KUKA KRL program: EPS_2_251729_MH1_A_20251114081654.src

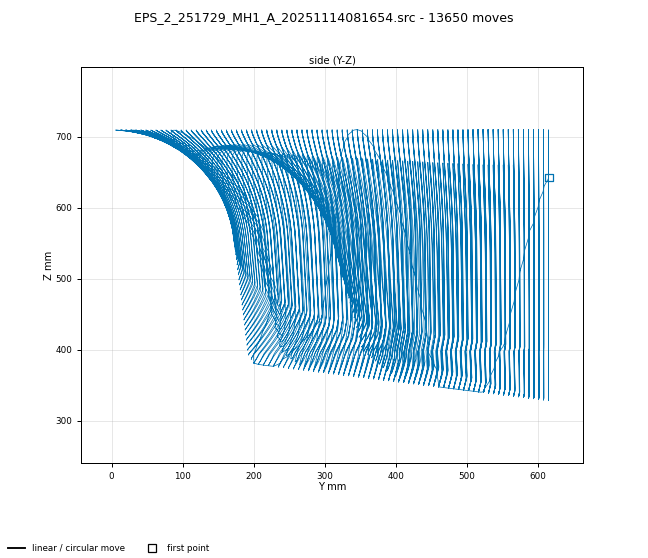
[picture p0: tool path of EPS_2_251729_MH1_A_20251114081654.src, 13650 of 13652 moves have a stored position in this frame; points joined in program order, loops and branches not executed]
&ACCESS RVP
&REL 4
&COMMENT QRS 19112012
&PARAM EDITMASK = *
DEF PART()
EXT BAS (BAS_COMMAND :IN,REAL :IN )
INT I
BAS (#INITMOV,0 )

;KUKA QRS Post kuka4.cps  Date:22-06-2017 !

File_ID=2915

QRS_PRE_INIT()

;Init var - Until changes are made in qrs_pre_init
Outlet_Square_prg=0
Inlet_1_Square_prg=0
Inlet_2_Square_prg=0
Inlet_3_Square_prg=0
Inlet_4_Square_prg=0
Inlet_5_Square_prg=0

Outlet_1={X 0.000, Y 517.920, Z 561.000, B 0.000, E1 0.000 }
Inlet_1={X 0.000, Y 525.500, Z 535.000, B 0.000, E1 90.000 }
Inlet_2={X 0.000, Y 517.920, Z 561.000, B 0.000, E1 180.000 }
Outlet_1_type=299
Inlet_1_type=251
Inlet_2_type=299
;QRS#1=Sidecore dimensions
;QRS#2=300-12" PVC SDR 35
;QRS#3=250-10" PVC SDR 35
;QRS#4=300-12" PVC SDR 35
;QRS#5=
;QRS#6=
;QRS#7=
;QRS#8=
;QRS#9=16M PSX
;QRS#10=14M PSX
;QRS#11=16M PSX
;QRS#12=
;QRS#13=
;QRS#14=
;QRS#15=
;QRS#16=1220x127x991 3,25'
;QRS#17=EPS Height
;QRS#18=710,5
;QRS#19=*
;QRS#20= UPDATED VERSION 22-06-2017
;QRS#21=*
Outlet_Square=0150
Inlet_1_Square=0100
Inlet_2_Square=0150
Inlet_3_Square=0
Inlet_4_Square=0
Inlet_5_Square=0
Mill_Square=1
Outlet_Square_Prg=206
Inlet_1_Square_prg=205
Inlet_2_Square_prg=206

QRS_INIT()

$ADVANCE=5

; T1
PTP {E1 173.418,E2 173.418}
PTP {X 0,Y 615.494,A -85,B 0,C 180,E1 173.418,E2 173.418,E3 0,E4 0,E5 0,E6 0}
QRS_SPEED_INIT()
LIN {X 0,Y 615.494,Z 642.738,A -85,B 0,C 180,E1 173.418,E2 173.418,E3 0,E4 0,E5 0,E6 0} C_VEL
LIN {X 0,Y 615.491,Z 635.744,A -85,B 0,C 180,E1 172.289,E2 172.289} C_VEL
LIN {X 0,Y 615.498,Z 628.27,A -85,B 0,C 180,E1 171.298,E2 171.298} C_VEL
LIN {X 0,Y 615.495,Z 619.291,A -85,B 0,C 180,E1 170.304,E2 170.304} C_VEL
LIN {X 0,Y 615.498,Z 608.204,A -85,B 0,C 180,E1 169.291,E2 169.291} C_VEL
LIN {X 0,Y 615.498,Z 597.279,A -85,B 0,C 180,E1 168.473,E2 168.473} C_VEL
LIN {X 0,Y 615.491,Z 584.981,A -85,B 0,C 180,E1 167.721,E2 167.721} C_VEL
LIN {X 0,Y 615.488,Z 573.143,A -85,B 0,C 180,E1 167.134,E2 167.134} C_VEL
LIN {X 0,Y 615.493,Z 560.215,A -85,B 0,C 180,E1 166.631,E2 166.631} C_VEL
LIN {X 0,Y 615.498,Z 547.234,A -85,B 0,C 180,E1 166.252,E2 166.252} C_VEL
LIN {X 0,Y 615.497,Z 533.996,A -85,B 0,C 180,E1 165.988,E2 165.988} C_VEL
LIN {X 0,Y 615.488,Z 397.614,A -85,B 0,C 180,E1 164.35,E2 164.35} C_VEL
LIN {X 0,Y 615.497,Z 392.889,A -85,B 0,C 180,E1 163.832,E2 163.832} C_VEL
LIN {X 0,Y 615.476,Z 369.093,A -85,B 0,C 180,E1 161.008,E2 161.008} C_VEL
LIN {X 0,Y 615.493,Z 345.922,A -85,B 0,C 180,E1 158.216,E2 158.216} C_VEL
LIN {X 0,Y 615.496,Z 328.786,A -85,B 0,C 180,E1 156.104,E2 156.104} C_VEL
LIN {X 0,Y 615.498,Z 328.434,A -85,B 0,C 180,E1 155.99,E2 155.99} C_VEL
LIN {X 0,Y 615.443,Z 328.325,A -85,B 0,C 180,E1 153.554,E2 153.554} C_VEL
LIN {X 0,Y 615.424,Z 328.324,A -85,B 0,C 180,E1 151.339,E2 151.339} C_VEL
LIN {X 0,Y 615.412,Z 328.324,A -85,B 0,C 180,E1 148.926,E2 148.926} C_VEL
LIN {X 0,Y 615.435,Z 328.323,A -85,B 0,C 180,E1 146.474,E2 146.474} C_VEL
LIN {X 0,Y 615.446,Z 328.325,A -85,B 0,C 180,E1 143.572,E2 143.572} C_VEL
LIN {X 0,Y 615.413,Z 328.324,A -85,B 0,C 180,E1 141.09,E2 141.09} C_VEL
LIN {X 0,Y 615.412,Z 328.324,A -85,B 0,C 180,E1 138.914,E2 138.914} C_VEL
LIN {X 0,Y 615.417,Z 328.324,A -85,B 0,C 180,E1 136.749,E2 136.749} C_VEL
LIN {X 0,Y 615.475,Z 328.323,A -85,B 0,C 180,E1 134.151,E2 134.151} C_VEL
LIN {X 0,Y 615.436,Z 328.324,A -85,B 0,C 180,E1 131.478,E2 131.478} C_VEL
LIN {X 0,Y 615.413,Z 328.324,A -85,B 0,C 180,E1 129.053,E2 129.053} C_VEL
LIN {X 0,Y 615.412,Z 328.324,A -85,B 0,C 180,E1 126.927,E2 126.927} C_VEL
LIN {X 0,Y 615.42,Z 328.324,A -85,B 0,C 180,E1 124.691,E2 124.691} C_VEL
LIN {X 0,Y 615.451,Z 328.323,A -85,B 0,C 180,E1 122.325,E2 122.325} C_VEL
LIN {X 0,Y 615.43,Z 328.324,A -85,B 0,C 180,E1 119.409,E2 119.409} C_VEL
LIN {X 0,Y 615.413,Z 328.324,A -85,B 0,C 180,E1 117.031,E2 117.031} C_VEL
LIN {X 0,Y 615.495,Z 328.571,A -85,B 0,C 180,E1 115.806,E2 115.806} C_VEL
LIN {X 0,Y 615.452,Z 348.722,A -85,B 0,C 180,E1 113.558,E2 113.558} C_VEL
LIN {X 0,Y 615.448,Z 371.548,A -85,B 0,C 180,E1 111.082,E2 111.082} C_VEL
LIN {X 0,Y 615.493,Z 396.288,A -85,B 0,C 180,E1 108.443,E2 108.443} C_VEL
LIN {X 0,Y 615.489,Z 398.972,A -85,B 0,C 180,E1 108.2,E2 108.2} C_VEL
LIN {X 0,Y 615.498,Z 565.217,A -85,B 0,C 180,E1 106.186,E2 106.186} C_VEL
LIN {X 0,Y 615.49,Z 580.613,A -85,B 0,C 180,E1 105.863,E2 105.863} C_VEL
LIN {X 0,Y 615.48,Z 595.975,A -85,B 0,C 180,E1 105.396,E2 105.396} C_VEL
LIN {X 0,Y 615.486,Z 610.66,A -85,B 0,C 180,E1 104.803,E2 104.803} C_VEL
LIN {X 0,Y 615.493,Z 624.629,A -85,B 0,C 180,E1 104.09,E2 104.09} C_VEL
LIN {X 0,Y 615.498,Z 637.489,A -85,B 0,C 180,E1 103.285,E2 103.285} C_VEL
LIN {X 0,Y 615.496,Z 649.742,A -85,B 0,C 180,E1 102.363,E2 102.363} C_VEL
LIN {X 0,Y 615.498,Z 660.897,A -85,B 0,C 180,E1 101.36,E2 101.36} C_VEL
LIN {X 0,Y 615.498,Z 671.702,A -85,B 0,C 180,E1 100.194,E2 100.194} C_VEL
LIN {X 0,Y 615.495,Z 680.684,A -85,B 0,C 180,E1 99.033,E2 99.033} C_VEL
LIN {X 0,Y 615.496,Z 688.117,A -85,B 0,C 180,E1 97.876,E2 97.876} C_VEL
LIN {X 0,Y 615.492,Z 695.052,A -85,B 0,C 180,E1 96.557,E2 96.557} C_VEL
LIN {X 0,Y 615.489,Z 700.498,A -85,B 0,C 180,E1 95.241,E2 95.241} C_VEL
LIN {X 0,Y 615.496,Z 704.619,A -85,B 0,C 180,E1 93.929,E2 93.929} C_VEL
LIN {X 0,Y 615.493,Z 707.525,A -85,B 0,C 180,E1 92.618,E2 92.618} C_VEL
LIN {X 0,Y 615.491,Z 709.276,A -85,B 0,C 180,E1 91.309,E2 91.309} C_VEL
LIN {X 0,Y 615.492,Z 709.884,A -85,B 0,C 180,E1 90,E2 90} C_VEL
LIN {X 0,Y 615.493,Z 709.338,A -85,B 0,C 180,E1 88.692,E2 88.692} C_VEL
LIN {X 0,Y 615.496,Z 707.675,A -85,B 0,C 180,E1 87.382,E2 87.382} C_VEL
LIN {X 0,Y 615.496,Z 704.861,A -85,B 0,C 180,E1 86.072,E2 86.072} C_VEL
LIN {X 0,Y 615.489,Z 700.835,A -85,B 0,C 180,E1 84.759,E2 84.759} C_VEL
LIN {X 0,Y 615.491,Z 695.378,A -85,B 0,C 180,E1 83.42,E2 83.42} C_VEL
LIN {X 0,Y 615.493,Z 688.661,A -85,B 0,C 180,E1 82.125,E2 82.125} C_VEL
LIN {X 0,Y 615.491,Z 680.145,A -85,B 0,C 180,E1 80.801,E2 80.801} C_VEL
LIN {X 0,Y 615.495,Z 671.067,A -85,B 0,C 180,E1 79.64,E2 79.64} C_VEL
LIN {X 0,Y 615.496,Z 661.792,A -85,B 0,C 180,E1 78.64,E2 78.64} C_VEL
LIN {X 0,Y 615.496,Z 649.823,A -85,B 0,C 180,E1 77.554,E2 77.554} C_VEL
LIN {X 0,Y 615.497,Z 637.582,A -85,B 0,C 180,E1 76.631,E2 76.631} C_VEL
LIN {X 0,Y 615.497,Z 624.88,A -85,B 0,C 180,E1 75.835,E2 75.835} C_VEL
LIN {X 0,Y 615.484,Z 610.782,A -85,B 0,C 180,E1 75.113,E2 75.113} C_VEL
LIN {X 0,Y 615.479,Z 596.123,A -85,B 0,C 180,E1 74.519,E2 74.519} C_VEL
LIN {X 0,Y 615.492,Z 581.162,A -85,B 0,C 180,E1 74.062,E2 74.062} C_VEL
LIN {X 0,Y 615.499,Z 565.657,A -85,B 0,C 180,E1 73.732,E2 73.732} C_VEL
LIN {X 0,Y 615.476,Z 447.644,A -85,B 0,C 180,E1 72.301,E2 72.301} C_VEL
LIN {X 0,Y 615.489,Z 398.701,A -85,B 0,C 180,E1 71.699,E2 71.699} C_VEL
LIN {X 0,Y 615.468,Z 374.018,A -85,B 0,C 180,E1 69.094,E2 69.094} C_VEL
LIN {X 0,Y 615.447,Z 351.178,A -85,B 0,C 180,E1 66.62,E2 66.62} C_VEL
LIN {X 0,Y 615.495,Z 328.663,A -85,B 0,C 180,E1 64.126,E2 64.126} C_VEL
LIN {X 0,Y 615.492,Z 328.327,A -85,B 0,C 180,E1 63.921,E2 63.921} C_VEL
LIN {X 0,Y 615.42,Z 328.325,A -85,B 0,C 180,E1 61.339,E2 61.339} C_VEL
LIN {X 0,Y 615.41,Z 328.325,A -85,B 0,C 180,E1 58.926,E2 58.926} C_VEL
LIN {X 0,Y 615.439,Z 328.325,A -85,B 0,C 180,E1 56.473,E2 56.473} C_VEL
LIN {X 0,Y 615.441,Z 328.323,A -85,B 0,C 180,E1 53.572,E2 53.572} C_VEL
LIN {X 0,Y 615.416,Z 328.323,A -85,B 0,C 180,E1 51.09,E2 51.09} C_VEL
LIN {X 0,Y 615.418,Z 328.324,A -85,B 0,C 180,E1 48.913,E2 48.913} C_VEL
LIN {X 0,Y 615.429,Z 328.323,A -85,B 0,C 180,E1 46.75,E2 46.75} C_VEL
LIN {X 0,Y 615.486,Z 328.322,A -85,B 0,C 180,E1 43.997,E2 43.997} C_VEL
LIN {X 0,Y 615.438,Z 328.32,A -85,B 0,C 180,E1 41.478,E2 41.478} C_VEL
LIN {X 0,Y 615.464,Z 328.319,A -85,B 0,C 180,E1 39.752,E2 39.752} C_VEL
LIN {X 0,Y 615.429,Z 328.32,A -85,B 0,C 180,E1 37.246,E2 37.246} C_VEL
LIN {X 0,Y 615.447,Z 328.323,A -85,B 0,C 180,E1 34.695,E2 34.695} C_VEL
LIN {X 0,Y 615.46,Z 328.317,A -85,B 0,C 180,E1 31.687,E2 31.687} C_VEL
LIN {X 0,Y 615.44,Z 328.318,A -85,B 0,C 180,E1 29.409,E2 29.409} C_VEL
LIN {X 0,Y 615.437,Z 328.32,A -85,B 0,C 180,E1 27.036,E2 27.036} C_VEL
LIN {X 0,Y 615.493,Z 328.324,A -85,B 0,C 180,E1 24.272,E2 24.272} C_VEL
LIN {X 0,Y 615.445,Z 328.317,A -85,B 0,C 180,E1 21.434,E2 21.434} C_VEL
LIN {X 0,Y 615.443,Z 328.317,A -85,B 0,C 180,E1 19.339,E2 19.339} C_VEL
LIN {X 0,Y 615.443,Z 328.318,A -85,B 0,C 180,E1 17.272,E2 17.272} C_VEL
LIN {X 0,Y 615.486,Z 328.324,A -85,B 0,C 180,E1 14.549,E2 14.549} C_VEL
LIN {X 0,Y 615.482,Z 328.312,A -85,B 0,C 180,E1 11.861,E2 11.861} C_VEL
LIN {X 0,Y 615.448,Z 328.318,A -85,B 0,C 180,E1 9.199,E2 9.199} C_VEL
LIN {X 0,Y 615.49,Z 328.326,A -85,B 0,C 180,E1 6.557,E2 6.557} C_VEL
LIN {X 0,Y 615.484,Z 328.311,A -85,B 0,C 180,E1 3.929,E2 3.929} C_VEL
LIN {X 0,Y 615.453,Z 328.316,A -85,B 0,C 180,E1 1.309,E2 1.309} C_VEL
LIN {X 0,Y 615.489,Z 328.324,A -85,B 0,C 180,E1 -1.309,E2 -1.309} C_VEL
LIN {X 0,Y 615.49,Z 328.311,A -85,B 0,C 180,E1 -3.928,E2 -3.928} C_VEL
LIN {X 0,Y 615.459,Z 328.314,A -85,B 0,C 180,E1 -6.557,E2 -6.557} C_VEL
LIN {X 0,Y 615.486,Z 328.323,A -85,B 0,C 180,E1 -9.199,E2 -9.199} C_VEL
LIN {X 0,Y 615.493,Z 328.31,A -85,B 0,C 180,E1 -11.861,E2 -11.861} C_VEL
LIN {X 0,Y 615.463,Z 328.314,A -85,B 0,C 180,E1 -14.55,E2 -14.55} C_VEL
LIN {X 0,Y 615.495,Z 328.326,A -85,B 0,C 180,E1 -17.27,E2 -17.27} C_VEL
LIN {X 0,Y 615.487,Z 328.308,A -85,B 0,C 180,E1 -20.033,E2 -20.033} C_VEL
LIN {X 0,Y 615.472,Z 328.319,A -85,B 0,C 180,E1 -22.845,E2 -22.845} C_VEL
LIN {X 0,Y 615.484,Z 328.316,A -85,B 0,C 180,E1 -25.568,E2 -25.568} C_VEL
LIN {X 0,Y 615.486,Z 328.309,A -85,B 0,C 180,E1 -27.915,E2 -27.915} C_VEL
LIN {X 0,Y 615.486,Z 328.308,A -85,B 0,C 180,E1 -30.16,E2 -30.16} C_VEL
LIN {X 0,Y 615.473,Z 328.313,A -85,B 0,C 180,E1 -32.458,E2 -32.458} C_VEL
LIN {X 0,Y 615.475,Z 328.321,A -85,B 0,C 180,E1 -34.816,E2 -34.816} C_VEL
LIN {X 0,Y 615.484,Z 328.322,A -85,B 0,C 180,E1 -37.242,E2 -37.242} C_VEL
LIN {X 0,Y 615.492,Z 328.306,A -85,B 0,C 180,E1 -40.09,E2 -40.09} C_VEL
LIN {X 0,Y 615.489,Z 328.326,A -85,B 0,C 180,E1 -43.047,E2 -43.047} C_VEL
LIN {X 0,Y 615.487,Z 328.307,A -85,B 0,C 180,E1 -46.003,E2 -46.003} C_VEL
LIN {X 0,Y 615.487,Z 328.326,A -85,B 0,C 180,E1 -48.905,E2 -48.905} C_VEL
LIN {X 0,Y 615.486,Z 328.322,A -85,B 0,C 180,E1 -51.096,E2 -51.096} C_VEL
LIN {X 0,Y 615.474,Z 328.313,A -85,B 0,C 180,E1 -53.574,E2 -53.574} C_VEL
LIN {X 0,Y 615.482,Z 328.316,A -85,B 0,C 180,E1 -56.466,E2 -56.466} C_VEL
LIN {X 0,Y 615.479,Z 328.322,A -85,B 0,C 180,E1 -59.08,E2 -59.08} C_VEL
LIN {X 0,Y 615.47,Z 328.313,A -85,B 0,C 180,E1 -61.553,E2 -61.553} C_VEL
LIN {X 0,Y 615.483,Z 328.313,A -85,B 0,C 180,E1 -64.284,E2 -64.284} C_VEL
LIN {X 0,Y 615.498,Z 328.586,A -85,B 0,C 180,E1 -64.937,E2 -64.937} C_VEL
LIN {X 0,Y 615.476,Z 347.018,A -85,B 0,C 180,E1 -66.8,E2 -66.8} C_VEL
LIN {X 0,Y 615.435,Z 372.213,A -85,B 0,C 180,E1 -69.267,E2 -69.267} C_VEL
LIN {X 0,Y 615.496,Z 398.105,A -85,B 0,C 180,E1 -71.742,E2 -71.742} C_VEL
LIN {X 0,Y 615.498,Z 564.923,A -85,B 0,C 180,E1 -73.764,E2 -73.764} C_VEL
LIN {X 0,Y 615.49,Z 580.716,A -85,B 0,C 180,E1 -74.095,E2 -74.095} C_VEL
LIN {X 0,Y 615.477,Z 596.053,A -85,B 0,C 180,E1 -74.562,E2 -74.562} C_VEL
LIN {X 0,Y 615.486,Z 609.755,A -85,B 0,C 180,E1 -75.113,E2 -75.113} C_VEL
LIN {X 0,Y 615.493,Z 624.047,A -85,B 0,C 180,E1 -75.834,E2 -75.834} C_VEL
LIN {X 0,Y 615.497,Z 636.9,A -85,B 0,C 180,E1 -76.631,E2 -76.631} C_VEL
LIN {X 0,Y 615.495,Z 649.256,A -85,B 0,C 180,E1 -77.554,E2 -77.554} C_VEL
LIN {X 0,Y 615.495,Z 659.607,A -85,B 0,C 180,E1 -78.473,E2 -78.473} C_VEL
LIN {X 0,Y 615.494,Z 669.185,A -85,B 0,C 180,E1 -79.473,E2 -79.473} C_VEL
LIN {X 0,Y 615.493,Z 678.578,A -85,B 0,C 180,E1 -80.636,E2 -80.636} C_VEL
LIN {X 0,Y 615.497,Z 686.381,A -85,B 0,C 180,E1 -81.794,E2 -81.794} C_VEL
LIN {X 0,Y 615.494,Z 693.609,A -85,B 0,C 180,E1 -83.102,E2 -83.102} C_VEL
LIN {X 0,Y 615.499,Z 699.437,A -85,B 0,C 180,E1 -84.43,E2 -84.43} C_VEL
LIN {X 0,Y 615.491,Z 702.86,A -85,B 0,C 180,E1 -85.416,E2 -85.416} C_VEL
LIN {X 0,Y 615.493,Z 706.318,A -85,B 0,C 180,E1 -86.727,E2 -86.727} C_VEL
LIN {X 0,Y 615.499,Z 708.593,A -85,B 0,C 180,E1 -88.037,E2 -88.037} C_VEL
LIN {X 0,Y 615.491,Z 709.741,A -85,B 0,C 180,E1 -89.346,E2 -89.346} C_VEL
LIN {X 0,Y 615.491,Z 709.741,A -85,B 0,C 180,E1 -90.654,E2 -90.654} C_VEL
LIN {X 0,Y 615.499,Z 708.593,A -85,B 0,C 180,E1 -91.963,E2 -91.963} C_VEL
LIN {X 0,Y 615.493,Z 706.318,A -85,B 0,C 180,E1 -93.273,E2 -93.273} C_VEL
LIN {X 0,Y 615.491,Z 702.86,A -85,B 0,C 180,E1 -94.585,E2 -94.585} C_VEL
LIN {X 0,Y 615.497,Z 698.142,A -85,B 0,C 180,E1 -95.899,E2 -95.899} C_VEL
LIN {X 0,Y 615.492,Z 692.029,A -85,B 0,C 180,E1 -97.216,E2 -97.216} C_VEL
LIN {X 0,Y 615.49,Z 684.332,A -85,B 0,C 180,E1 -98.537,E2 -98.537} C_VEL
LIN {X 0,Y 615.495,Z 676.113,A -85,B 0,C 180,E1 -99.696,E2 -99.696} C_VEL
LIN {X 0,Y 615.496,Z 665.899,A -85,B 0,C 180,E1 -100.892,E2 -100.892} C_VEL
LIN {X 0,Y 615.496,Z 656.066,A -85,B 0,C 180,E1 -101.861,E2 -101.861} C_VEL
LIN {X 0,Y 615.497,Z 643.946,A -85,B 0,C 180,E1 -102.865,E2 -102.865} C_VEL
LIN {X 0,Y 615.498,Z 631.796,A -85,B 0,C 180,E1 -103.706,E2 -103.706} C_VEL
LIN {X 0,Y 615.48,Z 618.377,A -85,B 0,C 180,E1 -104.473,E2 -104.473} C_VEL
LIN {X 0,Y 615.491,Z 603.845,A -85,B 0,C 180,E1 -105.141,E2 -105.141} C_VEL
LIN {X 0,Y 615.478,Z 589.612,A -85,B 0,C 180,E1 -105.651,E2 -105.651} C_VEL
LIN {X 0,Y 615.5,Z 575.075,A -85,B 0,C 180,E1 -106.037,E2 -106.037} C_VEL
LIN {X 0,Y 615.498,Z 560.297,A -85,B 0,C 180,E1 -106.301,E2 -106.301} C_VEL
LIN {X 0,Y 615.495,Z 398.102,A -85,B 0,C 180,E1 -108.258,E2 -108.258} C_VEL
LIN {X 0,Y 615.435,Z 372.211,A -85,B 0,C 180,E1 -110.733,E2 -110.733} C_VEL
LIN {X 0,Y 615.476,Z 347.016,A -85,B 0,C 180,E1 -113.201,E2 -113.201} C_VEL
LIN {X 0,Y 615.498,Z 328.586,A -85,B 0,C 180,E1 -115.063,E2 -115.063} C_VEL
LIN {X 0,Y 615.482,Z 328.314,A -85,B 0,C 180,E1 -115.716,E2 -115.716} C_VEL
LIN {X 0,Y 615.472,Z 328.314,A -85,B 0,C 180,E1 -118.448,E2 -118.448} C_VEL
LIN {X 0,Y 615.484,Z 328.327,A -85,B 0,C 180,E1 -121.086,E2 -121.086} C_VEL
LIN {X 0,Y 615.493,Z 328.307,A -85,B 0,C 180,E1 -124.022,E2 -124.022} C_VEL
LIN {X 0,Y 615.483,Z 328.326,A -85,B 0,C 180,E1 -126.936,E2 -126.936} C_VEL
LIN {X 0,Y 615.475,Z 328.311,A -85,B 0,C 180,E1 -129.751,E2 -129.751} C_VEL
LIN {X 0,Y 615.489,Z 328.316,A -85,B 0,C 180,E1 -132.353,E2 -132.353} C_VEL
LIN {X 0,Y 615.463,Z 328.32,A -85,B 0,C 180,E1 -135.071,E2 -135.071} C_VEL
LIN {X 0,Y 615.487,Z 328.311,A -85,B 0,C 180,E1 -137.92,E2 -137.92} C_VEL
LIN {X 0,Y 615.491,Z 328.319,A -85,B 0,C 180,E1 -140.25,E2 -140.25} C_VEL
LIN {X 0,Y 615.444,Z 328.32,A -85,B 0,C 180,E1 -143.069,E2 -143.069} C_VEL
LIN {X 0,Y 615.439,Z 328.319,A -85,B 0,C 180,E1 -145.306,E2 -145.306} C_VEL
LIN {X 0,Y 615.457,Z 328.318,A -85,B 0,C 180,E1 -147.674,E2 -147.674} C_VEL
LIN {X 0,Y 615.447,Z 328.324,A -85,B 0,C 180,E1 -150.592,E2 -150.592} C_VEL
LIN {X 0,Y 615.421,Z 328.323,A -85,B 0,C 180,E1 -152.967,E2 -152.967} C_VEL
LIN {X 0,Y 615.416,Z 328.324,A -85,B 0,C 180,E1 -155.005,E2 -155.005} C_VEL
LIN {X 0,Y 615.491,Z 328.47,A -85,B 0,C 180,E1 -156.105,E2 -156.105} C_VEL
LIN {X 0,Y 615.494,Z 328.899,A -85,B 0,C 180,E1 -156.218,E2 -156.218} C_VEL
LIN {X 0,Y 615.48,Z 350.974,A -85,B 0,C 180,E1 -158.919,E2 -158.919} C_VEL
LIN {X 0,Y 615.499,Z 374.313,A -85,B 0,C 180,E1 -161.722,E2 -161.722} C_VEL
LIN {X 0,Y 615.485,Z 397.189,A -85,B 0,C 180,E1 -164.413,E2 -164.413} C_VEL
LIN {X 0,Y 615.486,Z 399.616,A -85,B 0,C 180,E1 -164.477,E2 -164.477} C_VEL
LIN {X 0,Y 615.498,Z 535.161,A -85,B 0,C 180,E1 -166.095,E2 -166.095} C_VEL
LIN {X 0,Y 615.497,Z 548.75,A -85,B 0,C 180,E1 -166.379,E2 -166.379} C_VEL
LIN {X 0,Y 615.495,Z 562.489,A -85,B 0,C 180,E1 -166.799,E2 -166.799} C_VEL
LIN {X 0,Y 615.49,Z 574.901,A -85,B 0,C 180,E1 -167.302,E2 -167.302} C_VEL
LIN {X 0,Y 615.498,Z 587.842,A -85,B 0,C 180,E1 -167.972,E2 -167.972} C_VEL
LIN {X 0,Y 615.499,Z 599.559,A -85,B 0,C 180,E1 -168.724,E2 -168.724} C_VEL
LIN {X 0,Y 615.498,Z 611.226,A -85,B 0,C 180,E1 -169.64,E2 -169.64} C_VEL
LIN {X 0,Y 615.497,Z 621.651,A -85,B 0,C 180,E1 -170.636,E2 -170.636} C_VEL
LIN {X 0,Y 615.496,Z 630.24,A -85,B 0,C 180,E1 -171.629,E2 -171.629} C_VEL
LIN {X 0,Y 615.495,Z 638.453,A -85,B 0,C 180,E1 -172.784,E2 -172.784} C_VEL
LIN {X 0,Y 615.496,Z 644.184,A -85,B 0,C 180,E1 -173.773,E2 -173.773} C_VEL
LIN {X 0,Y 615.494,Z 648.887,A -85,B 0,C 180,E1 -174.759,E2 -174.759} C_VEL
LIN {X 0,Y 615.496,Z 653.757,A -85,B 0,C 180,E1 -176.072,E2 -176.072} C_VEL
LIN {X 0,Y 615.496,Z 657.154,A -85,B 0,C 180,E1 -177.382,E2 -177.382} C_VEL
LIN {X 0,Y 615.493,Z 659.174,A -85,B 0,C 180,E1 -178.691,E2 -178.691} C_VEL
LIN {X 0,Y 615.494,Z 659.884,A -85,B 0,C 180,E1 -180,E2 -180} C_VEL
LIN {X 0,Y 615.49,Z 659.28,A -85,B 0,C 180,E1 -181.309,E2 -181.309} C_VEL
LIN {X 0,Y 615.493,Z 657.35,A -85,B 0,C 180,E1 -182.618,E2 -182.618} C_VEL
LIN {X 0,Y 615.496,Z 654.045,A -85,B 0,C 180,E1 -183.929,E2 -183.929} C_VEL
LIN {X 0,Y 615.496,Z 649.273,A -85,B 0,C 180,E1 -185.241,E2 -185.241} C_VEL
LIN {X 0,Y 615.495,Z 642.874,A -85,B 0,C 180,E1 -186.557,E2 -186.557} C_VEL
LIN {X 0,Y 615.494,Z 642.738,A -85,B 0,C 180,E1 -186.582,E2 -186.582} C_VEL
LIN {X 0,Y 614.823,Z 640.104,A -85,B 0,C 180,E1 -187.065,E2 -187.065} C_VEL
LIN {X 0,Y 611.977,Z 635.518,A -85,B 0,C 180,E1 -187.841,E2 -187.841} C_VEL
LIN {X 0,Y 609.129,Z 630.273,A -85,B 0,C 180,E1 -188.592,E2 -188.592} C_VEL
LIN {X 0,Y 608.47,Z 626.658,A -85,B 0,C 180,E1 -189.033,E2 -189.033} C_VEL
LIN {X 0,Y 608.472,Z 617.861,A -85,B 0,C 180,E1 -189.977,E2 -189.977} C_VEL
LIN {X 0,Y 608.506,Z 606.618,A -85,B 0,C 180,E1 -190.973,E2 -190.973} C_VEL
LIN {X 0,Y 608.535,Z 594.824,A -85,B 0,C 180,E1 -191.829,E2 -191.829} C_VEL
LIN {X 0,Y 608.529,Z 581.908,A -85,B 0,C 180,E1 -192.591,E2 -192.591} C_VEL
LIN {X 0,Y 608.566,Z 568.231,A -85,B 0,C 180,E1 -193.227,E2 -193.227} C_VEL
LIN {X 0,Y 608.607,Z 555.002,A -85,B 0,C 180,E1 -193.694,E2 -193.694} C_VEL
LIN {X 0,Y 608.624,Z 540.476,A -85,B 0,C 180,E1 -194.057,E2 -194.057} C_VEL
LIN {X 0,Y 608.632,Z 525.252,A -85,B 0,C 180,E1 -194.289,E2 -194.289} C_VEL
LIN {X 0,Y 608.58,Z 397.863,A -85,B 0,C 180,E1 -195.822,E2 -195.822} C_VEL
LIN {X 0,Y 608.517,Z 396.622,A -85,B 0,C 180,E1 -195.92,E2 -195.92} C_VEL
LIN {X 0,Y 608.533,Z 373.11,A -85,B 0,C 180,E1 -198.732,E2 -198.732} C_VEL
LIN {X 0,Y 608.598,Z 350.263,A -85,B 0,C 180,E1 -201.509,E2 -201.509} C_VEL
LIN {X 0,Y 608.594,Z 330.064,A -85,B 0,C 180,E1 -204.01,E2 -204.01} C_VEL
LIN {X 0,Y 608.481,Z 329.416,A -85,B 0,C 180,E1 -204.153,E2 -204.153} C_VEL
LIN {X 0,Y 608.389,Z 329.321,A -85,B 0,C 180,E1 -206.777,E2 -206.777} C_VEL
LIN {X 0,Y 608.386,Z 329.32,A -85,B 0,C 180,E1 -209.024,E2 -209.024} C_VEL
LIN {X 0,Y 608.391,Z 329.321,A -85,B 0,C 180,E1 -211.321,E2 -211.321} C_VEL
LIN {X 0,Y 608.426,Z 329.321,A -85,B 0,C 180,E1 -213.728,E2 -213.728} C_VEL
LIN {X 0,Y 608.437,Z 329.325,A -85,B 0,C 180,E1 -216.093,E2 -216.093} C_VEL
LIN {X 0,Y 608.394,Z 329.322,A -85,B 0,C 180,E1 -218.594,E2 -218.594} C_VEL
LIN {X 0,Y 608.434,Z 329.32,A -85,B 0,C 180,E1 -220.327,E2 -220.327} C_VEL
LIN {X 0,Y 608.428,Z 329.321,A -85,B 0,C 180,E1 -222.331,E2 -222.331} C_VEL
LIN {X 0,Y 608.398,Z 329.32,A -85,B 0,C 180,E1 -224.801,E2 -224.801} C_VEL
LIN {X 0,Y 608.384,Z 329.32,A -85,B 0,C 180,E1 -227.034,E2 -227.034} C_VEL
LIN {X 0,Y 608.387,Z 329.321,A -85,B 0,C 180,E1 -228.818,E2 -228.818} C_VEL
LIN {X 0,Y 608.392,Z 329.321,A -85,B 0,C 180,E1 -231.406,E2 -231.406} C_VEL
LIN {X 0,Y 608.442,Z 329.323,A -85,B 0,C 180,E1 -233.955,E2 -233.955} C_VEL
LIN {X 0,Y 608.444,Z 329.319,A -85,B 0,C 180,E1 -236.328,E2 -236.328} C_VEL
LIN {X 0,Y 608.404,Z 329.319,A -85,B 0,C 180,E1 -238.739,E2 -238.739} C_VEL
LIN {X 0,Y 608.387,Z 329.321,A -85,B 0,C 180,E1 -240.976,E2 -240.976} C_VEL
LIN {X 0,Y 608.485,Z 329.424,A -85,B 0,C 180,E1 -243.966,E2 -243.966} C_VEL
LIN {X 0,Y 608.726,Z 333.074,A -85,B 0,C 180,E1 -244.418,E2 -244.418} C_VEL
LIN {X 0,Y 608.615,Z 356.881,A -85,B 0,C 180,E1 -247.062,E2 -247.062} C_VEL
LIN {X 0,Y 608.608,Z 382.966,A -85,B 0,C 180,E1 -249.907,E2 -249.907} C_VEL
LIN {X 0,Y 608.603,Z 398.536,A -85,B 0,C 180,E1 -251.566,E2 -251.566} C_VEL
LIN {X 0,Y 608.765,Z 403.562,A -85,B 0,C 180,E1 -251.653,E2 -251.653} C_VEL
LIN {X 0,Y 608.699,Z 565.25,A -85,B 0,C 180,E1 -253.629,E2 -253.629} C_VEL
LIN {X 0,Y 608.651,Z 580.634,A -85,B 0,C 180,E1 -253.954,E2 -253.954} C_VEL
LIN {X 0,Y 608.61,Z 595.973,A -85,B 0,C 180,E1 -254.426,E2 -254.426} C_VEL
LIN {X 0,Y 608.584,Z 610.657,A -85,B 0,C 180,E1 -255.025,E2 -255.025} C_VEL
LIN {X 0,Y 608.571,Z 624.436,A -85,B 0,C 180,E1 -255.735,E2 -255.735} C_VEL
LIN {X 0,Y 608.548,Z 637.545,A -85,B 0,C 180,E1 -256.56,E2 -256.56} C_VEL
LIN {X 0,Y 608.505,Z 649.836,A -85,B 0,C 180,E1 -257.493,E2 -257.493} C_VEL
LIN {X 0,Y 608.497,Z 661.046,A -85,B 0,C 180,E1 -258.508,E2 -258.508} C_VEL
LIN {X 0,Y 608.477,Z 671.931,A -85,B 0,C 180,E1 -259.687,E2 -259.687} C_VEL
LIN {X 0,Y 608.469,Z 680.979,A -85,B 0,C 180,E1 -260.862,E2 -260.862} C_VEL
LIN {X 0,Y 608.46,Z 688.478,A -85,B 0,C 180,E1 -262.033,E2 -262.033} C_VEL
LIN {X 0,Y 608.445,Z 695.629,A -85,B 0,C 180,E1 -263.397,E2 -263.397} C_VEL
LIN {X 0,Y 608.435,Z 700.994,A -85,B 0,C 180,E1 -264.698,E2 -264.698} C_VEL
LIN {X 0,Y 608.432,Z 705.166,A -85,B 0,C 180,E1 -266.026,E2 -266.026} C_VEL
LIN {X 0,Y 608.421,Z 708.11,A -85,B 0,C 180,E1 -267.352,E2 -267.352} C_VEL
LIN {X 0,Y 608.444,Z 709.881,A -85,B 0,C 180,E1 -268.676,E2 -268.676} C_VEL
LIN {X 0,Y 608.432,Z 710.495,A -85,B 0,C 180,E1 -270,E2 -270} C_VEL
LIN {X 0,Y 608.445,Z 709.945,A -85,B 0,C 180,E1 -271.324,E2 -271.324} C_VEL
LIN {X 0,Y 608.424,Z 708.26,A -85,B 0,C 180,E1 -272.648,E2 -272.648} C_VEL
LIN {X 0,Y 608.432,Z 705.407,A -85,B 0,C 180,E1 -273.974,E2 -273.974} C_VEL
LIN {X 0,Y 608.435,Z 701.33,A -85,B 0,C 180,E1 -275.302,E2 -275.302} C_VEL
LIN {X 0,Y 608.446,Z 695.922,A -85,B 0,C 180,E1 -276.633,E2 -276.633} C_VEL
LIN {X 0,Y 608.458,Z 689.021,A -85,B 0,C 180,E1 -277.967,E2 -277.967} C_VEL
LIN {X 0,Y 608.466,Z 681.592,A -85,B 0,C 180,E1 -279.138,E2 -279.138} C_VEL
LIN {X 0,Y 608.477,Z 672.661,A -85,B 0,C 180,E1 -280.313,E2 -280.313} C_VEL
LIN {X 0,Y 608.496,Z 661.949,A -85,B 0,C 180,E1 -281.492,E2 -281.492} C_VEL
LIN {X 0,Y 608.513,Z 649.902,A -85,B 0,C 180,E1 -282.591,E2 -282.591} C_VEL
LIN {X 0,Y 608.543,Z 637.621,A -85,B 0,C 180,E1 -283.525,E2 -283.525} C_VEL
LIN {X 0,Y 608.585,Z 624.675,A -85,B 0,C 180,E1 -284.342,E2 -284.342} C_VEL
LIN {X 0,Y 608.585,Z 610.758,A -85,B 0,C 180,E1 -285.06,E2 -285.06} C_VEL
LIN {X 0,Y 608.631,Z 596.089,A -85,B 0,C 180,E1 -285.659,E2 -285.659} C_VEL
LIN {X 0,Y 608.67,Z 580.52,A -85,B 0,C 180,E1 -286.138,E2 -286.138} C_VEL
LIN {X 0,Y 608.696,Z 565.068,A -85,B 0,C 180,E1 -286.464,E2 -286.464} C_VEL
LIN {X 0,Y 608.683,Z 399.384,A -85,B 0,C 180,E1 -288.492,E2 -288.492} C_VEL
LIN {X 0,Y 608.566,Z 398.143,A -85,B 0,C 180,E1 -288.556,E2 -288.556} C_VEL
LIN {X 0,Y 608.575,Z 374.013,A -85,B 0,C 180,E1 -291.154,E2 -291.154} C_VEL
LIN {X 0,Y 608.614,Z 352.804,A -85,B 0,C 180,E1 -293.478,E2 -293.478} C_VEL
LIN {X 0,Y 608.727,Z 331.079,A -85,B 0,C 180,E1 -295.897,E2 -295.897} C_VEL
LIN {X 0,Y 608.474,Z 329.367,A -85,B 0,C 180,E1 -296.149,E2 -296.149} C_VEL
LIN {X 0,Y 608.383,Z 329.321,A -85,B 0,C 180,E1 -299.024,E2 -299.024} C_VEL
LIN {X 0,Y 608.405,Z 329.32,A -85,B 0,C 180,E1 -301.32,E2 -301.32} C_VEL
LIN {X 0,Y 608.424,Z 329.323,A -85,B 0,C 180,E1 -303.728,E2 -303.728} C_VEL
LIN {X 0,Y 608.438,Z 329.322,A -85,B 0,C 180,E1 -306.093,E2 -306.093} C_VEL
LIN {X 0,Y 608.395,Z 329.321,A -85,B 0,C 180,E1 -308.594,E2 -308.594} C_VEL
LIN {X 0,Y 608.392,Z 329.321,A -85,B 0,C 180,E1 -311.182,E2 -311.182} C_VEL
LIN {X 0,Y 608.461,Z 329.322,A -85,B 0,C 180,E1 -313.87,E2 -313.87} C_VEL
LIN {X 0,Y 608.422,Z 329.316,A -85,B 0,C 180,E1 -316.696,E2 -316.696} C_VEL
LIN {X 0,Y 608.396,Z 329.319,A -85,B 0,C 180,E1 -318.818,E2 -318.818} C_VEL
LIN {X 0,Y 608.407,Z 329.322,A -85,B 0,C 180,E1 -321.407,E2 -321.407} C_VEL
LIN {X 0,Y 608.444,Z 329.321,A -85,B 0,C 180,E1 -323.955,E2 -323.955} C_VEL
LIN {X 0,Y 608.443,Z 329.315,A -85,B 0,C 180,E1 -326.328,E2 -326.328} C_VEL
LIN {X 0,Y 608.428,Z 329.315,A -85,B 0,C 180,E1 -328.735,E2 -328.735} C_VEL
LIN {X 0,Y 608.457,Z 329.317,A -85,B 0,C 180,E1 -331.383,E2 -331.383} C_VEL
LIN {X 0,Y 608.449,Z 329.314,A -85,B 0,C 180,E1 -334.284,E2 -334.284} C_VEL
LIN {X 0,Y 608.46,Z 329.314,A -85,B 0,C 180,E1 -336.155,E2 -336.155} C_VEL
LIN {X 0,Y 608.449,Z 329.314,A -85,B 0,C 180,E1 -338.308,E2 -338.308} C_VEL
LIN {X 0,Y 608.441,Z 329.317,A -85,B 0,C 180,E1 -341.13,E2 -341.13} C_VEL
LIN {X 0,Y 608.461,Z 329.316,A -85,B 0,C 180,E1 -343.906,E2 -343.906} C_VEL
LIN {X 0,Y 608.434,Z 329.315,A -85,B 0,C 180,E1 -346.643,E2 -346.643} C_VEL
LIN {X 0,Y 608.456,Z 329.319,A -85,B 0,C 180,E1 -349.35,E2 -349.35} C_VEL
LIN {X 0,Y 608.475,Z 329.312,A -85,B 0,C 180,E1 -352.033,E2 -352.033} C_VEL
LIN {X 0,Y 608.435,Z 329.315,A -85,B 0,C 180,E1 -354.698,E2 -354.698} C_VEL
LIN {X 0,Y 608.481,Z 329.318,A -85,B 0,C 180,E1 -357.352,E2 -357.352} C_VEL
LIN {X 0,Y 608.477,Z 329.311,A -85,B 0,C 180,E1 -360,E2 -360} C_VEL
LIN {X 0,Y 608.451,Z 329.313,A -85,B 0,C 180,E1 -362.648,E2 -362.648} C_VEL
LIN {X 0,Y 608.466,Z 329.32,A -85,B 0,C 180,E1 -365.302,E2 -365.302} C_VEL
LIN {X 0,Y 608.479,Z 329.31,A -85,B 0,C 180,E1 -367.967,E2 -367.967} C_VEL
LIN {X 0,Y 608.443,Z 329.315,A -85,B 0,C 180,E1 -370.65,E2 -370.65} C_VEL
LIN {X 0,Y 608.468,Z 329.32,A -85,B 0,C 180,E1 -373.356,E2 -373.356} C_VEL
LIN {X 0,Y 608.456,Z 329.312,A -85,B 0,C 180,E1 -376.094,E2 -376.094} C_VEL
LIN {X 0,Y 608.449,Z 329.317,A -85,B 0,C 180,E1 -378.87,E2 -378.87} C_VEL
LIN {X 0,Y 608.47,Z 329.313,A -85,B 0,C 180,E1 -381.691,E2 -381.691} C_VEL
LIN {X 0,Y 608.448,Z 329.314,A -85,B 0,C 180,E1 -384.571,E2 -384.571} C_VEL
LIN {X 0,Y 608.481,Z 329.319,A -85,B 0,C 180,E1 -387.208,E2 -387.208} C_VEL
LIN {X 0,Y 608.468,Z 329.31,A -85,B 0,C 180,E1 -389.972,E2 -389.972} C_VEL
LIN {X 0,Y 608.452,Z 329.319,A -85,B 0,C 180,E1 -392.88,E2 -392.88} C_VEL
LIN {X 0,Y 608.437,Z 329.322,A -85,B 0,C 180,E1 -395.278,E2 -395.278} C_VEL
LIN {X 0,Y 608.468,Z 329.311,A -85,B 0,C 180,E1 -397.746,E2 -397.746} C_VEL
LIN {X 0,Y 608.451,Z 329.313,A -85,B 0,C 180,E1 -400.329,E2 -400.329} C_VEL
LIN {X 0,Y 608.454,Z 329.322,A -85,B 0,C 180,E1 -402.96,E2 -402.96} C_VEL
LIN {X 0,Y 608.458,Z 329.312,A -85,B 0,C 180,E1 -405.736,E2 -405.736} C_VEL
LIN {X 0,Y 608.459,Z 329.317,A -85,B 0,C 180,E1 -408.658,E2 -408.658} C_VEL
LIN {X 0,Y 608.469,Z 329.313,A -85,B 0,C 180,E1 -411.412,E2 -411.412} C_VEL
LIN {X 0,Y 608.447,Z 329.313,A -85,B 0,C 180,E1 -413.954,E2 -413.954} C_VEL
LIN {X 0,Y 608.463,Z 329.313,A -85,B 0,C 180,E1 -416.329,E2 -416.329} C_VEL
LIN {X 0,Y 608.478,Z 329.318,A -85,B 0,C 180,E1 -418.728,E2 -418.728} C_VEL
LIN {X 0,Y 608.459,Z 329.314,A -85,B 0,C 180,E1 -421.382,E2 -421.382} C_VEL
LIN {X 0,Y 608.437,Z 329.316,A -85,B 0,C 180,E1 -423.964,E2 -423.964} C_VEL
LIN {X 0,Y 608.498,Z 329.481,A -85,B 0,C 180,E1 -424.724,E2 -424.724} C_VEL
LIN {X 0,Y 608.739,Z 332.621,A -85,B 0,C 180,E1 -425.077,E2 -425.077} C_VEL
LIN {X 0,Y 608.662,Z 359.615,A -85,B 0,C 180,E1 -427.781,E2 -427.781} C_VEL
LIN {X 0,Y 608.563,Z 388.409,A -85,B 0,C 180,E1 -430.609,E2 -430.609} C_VEL
LIN {X 0,Y 608.627,Z 398.103,A -85,B 0,C 180,E1 -431.529,E2 -431.529} C_VEL
LIN {X 0,Y 608.702,Z 510.075,A -85,B 0,C 180,E1 -432.899,E2 -432.899} C_VEL
LIN {X 0,Y 608.676,Z 565.864,A -85,B 0,C 180,E1 -433.594,E2 -433.594} C_VEL
LIN {X 0,Y 608.656,Z 581.491,A -85,B 0,C 180,E1 -433.933,E2 -433.933} C_VEL
LIN {X 0,Y 608.617,Z 596.051,A -85,B 0,C 180,E1 -434.383,E2 -434.383} C_VEL
LIN {X 0,Y 608.602,Z 609.758,A -85,B 0,C 180,E1 -434.94,E2 -434.94} C_VEL
LIN {X 0,Y 608.573,Z 623.238,A -85,B 0,C 180,E1 -435.624,E2 -435.624} C_VEL
LIN {X 0,Y 608.554,Z 635.665,A -85,B 0,C 180,E1 -436.39,E2 -436.39} C_VEL
LIN {X 0,Y 608.528,Z 648.284,A -85,B 0,C 180,E1 -437.324,E2 -437.324} C_VEL
LIN {X 0,Y 608.496,Z 659.748,A -85,B 0,C 180,E1 -438.339,E2 -438.339} C_VEL
LIN {X 0,Y 608.475,Z 669.389,A -85,B 0,C 180,E1 -439.35,E2 -439.35} C_VEL
LIN {X 0,Y 608.476,Z 678.854,A -85,B 0,C 180,E1 -440.527,E2 -440.527} C_VEL
LIN {X 0,Y 608.456,Z 686.73,A -85,B 0,C 180,E1 -441.699,E2 -441.699} C_VEL
LIN {X 0,Y 608.439,Z 694.088,A -85,B 0,C 180,E1 -443.034,E2 -443.034} C_VEL
LIN {X 0,Y 608.45,Z 699.924,A -85,B 0,C 180,E1 -444.366,E2 -444.366} C_VEL
LIN {X 0,Y 608.427,Z 703.383,A -85,B 0,C 180,E1 -445.362,E2 -445.362} C_VEL
LIN {X 0,Y 608.421,Z 706.886,A -85,B 0,C 180,E1 -446.689,E2 -446.689} C_VEL
LIN {X 0,Y 608.444,Z 709.191,A -85,B 0,C 180,E1 -448.014,E2 -448.014} C_VEL
LIN {X 0,Y 608.434,Z 710.351,A -85,B 0,C 180,E1 -449.338,E2 -449.338} C_VEL
LIN {X 0,Y 608.434,Z 710.351,A -85,B 0,C 180,E1 -450.662,E2 -450.662} C_VEL
LIN {X 0,Y 608.444,Z 709.191,A -85,B 0,C 180,E1 -451.986,E2 -451.986} C_VEL
LIN {X 0,Y 608.421,Z 706.885,A -85,B 0,C 180,E1 -453.311,E2 -453.311} C_VEL
LIN {X 0,Y 608.427,Z 703.382,A -85,B 0,C 180,E1 -454.638,E2 -454.638} C_VEL
LIN {X 0,Y 608.435,Z 698.607,A -85,B 0,C 180,E1 -455.967,E2 -455.967} C_VEL
LIN {X 0,Y 608.456,Z 692.425,A -85,B 0,C 180,E1 -457.3,E2 -457.3} C_VEL
LIN {X 0,Y 608.465,Z 684.653,A -85,B 0,C 180,E1 -458.636,E2 -458.636} C_VEL
LIN {X 0,Y 608.471,Z 676.369,A -85,B 0,C 180,E1 -459.809,E2 -459.809} C_VEL
LIN {X 0,Y 608.492,Z 665.651,A -85,B 0,C 180,E1 -461.063,E2 -461.063} C_VEL
LIN {X 0,Y 608.523,Z 654.273,A -85,B 0,C 180,E1 -462.168,E2 -462.168} C_VEL
LIN {X 0,Y 608.547,Z 642.852,A -85,B 0,C 180,E1 -463.1,E2 -463.1} C_VEL
LIN {X 0,Y 608.563,Z 630.445,A -85,B 0,C 180,E1 -463.95,E2 -463.95} C_VEL
LIN {X 0,Y 608.564,Z 616.856,A -85,B 0,C 180,E1 -464.718,E2 -464.718} C_VEL
LIN {X 0,Y 608.629,Z 602.788,A -85,B 0,C 180,E1 -465.359,E2 -465.359} C_VEL
LIN {X 0,Y 608.634,Z 588.297,A -85,B 0,C 180,E1 -465.874,E2 -465.874} C_VEL
LIN {X 0,Y 608.676,Z 572.925,A -85,B 0,C 180,E1 -466.272,E2 -466.272} C_VEL
LIN {X 0,Y 608.702,Z 557.273,A -85,B 0,C 180,E1 -466.531,E2 -466.531} C_VEL
LIN {X 0,Y 608.637,Z 398.248,A -85,B 0,C 180,E1 -468.466,E2 -468.466} C_VEL
LIN {X 0,Y 608.564,Z 388.407,A -85,B 0,C 180,E1 -469.392,E2 -469.392} C_VEL
LIN {X 0,Y 608.662,Z 359.614,A -85,B 0,C 180,E1 -472.219,E2 -472.219} C_VEL
LIN {X 0,Y 608.74,Z 332.619,A -85,B 0,C 180,E1 -474.923,E2 -474.923} C_VEL
LIN {X 0,Y 608.501,Z 329.48,A -85,B 0,C 180,E1 -475.276,E2 -475.276} C_VEL
LIN {X 0,Y 608.451,Z 329.317,A -85,B 0,C 180,E1 -477.518,E2 -477.518} C_VEL
LIN {X 0,Y 608.468,Z 329.311,A -85,B 0,C 180,E1 -479.972,E2 -479.972} C_VEL
LIN {X 0,Y 608.452,Z 329.322,A -85,B 0,C 180,E1 -482.88,E2 -482.88} C_VEL
LIN {X 0,Y 608.439,Z 329.319,A -85,B 0,C 180,E1 -485.278,E2 -485.278} C_VEL
LIN {X 0,Y 608.466,Z 329.311,A -85,B 0,C 180,E1 -487.747,E2 -487.747} C_VEL
LIN {X 0,Y 608.456,Z 329.316,A -85,B 0,C 180,E1 -490.329,E2 -490.329} C_VEL
LIN {X 0,Y 608.439,Z 329.32,A -85,B 0,C 180,E1 -492.961,E2 -492.961} C_VEL
LIN {X 0,Y 608.451,Z 329.313,A -85,B 0,C 180,E1 -495.737,E2 -495.737} C_VEL
LIN {X 0,Y 608.458,Z 329.32,A -85,B 0,C 180,E1 -498.658,E2 -498.658} C_VEL
LIN {X 0,Y 608.459,Z 329.313,A -85,B 0,C 180,E1 -501.761,E2 -501.761} C_VEL
LIN {X 0,Y 608.432,Z 329.32,A -85,B 0,C 180,E1 -504.722,E2 -504.722} C_VEL
LIN {X 0,Y 608.425,Z 329.317,A -85,B 0,C 180,E1 -507.119,E2 -507.119} C_VEL
LIN {X 0,Y 608.471,Z 329.318,A -85,B 0,C 180,E1 -510.028,E2 -510.028} C_VEL
LIN {X 0,Y 608.409,Z 329.32,A -85,B 0,C 180,E1 -512.806,E2 -512.806} C_VEL
LIN {X 0,Y 608.415,Z 329.32,A -85,B 0,C 180,E1 -515.427,E2 -515.427} C_VEL
LIN {X 0,Y 608.497,Z 329.479,A -85,B 0,C 180,E1 -515.968,E2 -515.968} C_VEL
LIN {X 0,Y 608.63,Z 332.158,A -85,B 0,C 180,E1 -516.343,E2 -516.343} C_VEL
LIN {X 0,Y 608.576,Z 353.874,A -85,B 0,C 180,E1 -519.023,E2 -519.023} C_VEL
LIN {X 0,Y 608.563,Z 377.039,A -85,B 0,C 180,E1 -521.832,E2 -521.832} C_VEL
LIN {X 0,Y 608.532,Z 397.518,A -85,B 0,C 180,E1 -524.252,E2 -524.252} C_VEL
LIN {X 0,Y 608.661,Z 408.603,A -85,B 0,C 180,E1 -524.406,E2 -524.406} C_VEL
LIN {X 0,Y 608.608,Z 535.991,A -85,B 0,C 180,E1 -525.949,E2 -525.949} C_VEL
LIN {X 0,Y 608.613,Z 550.31,A -85,B 0,C 180,E1 -526.264,E2 -526.264} C_VEL
LIN {X 0,Y 608.585,Z 563.648,A -85,B 0,C 180,E1 -526.689,E2 -526.689} C_VEL
LIN {X 0,Y 608.538,Z 576.702,A -85,B 0,C 180,E1 -527.24,E2 -527.24} C_VEL
LIN {X 0,Y 608.538,Z 589.345,A -85,B 0,C 180,E1 -527.917,E2 -527.917} C_VEL
LIN {X 0,Y 608.499,Z 600.848,A -85,B 0,C 180,E1 -528.677,E2 -528.677} C_VEL
LIN {X 0,Y 608.495,Z 611.415,A -85,B 0,C 180,E1 -529.519,E2 -529.519} C_VEL
LIN {X 0,Y 608.48,Z 621.899,A -85,B 0,C 180,E1 -530.527,E2 -530.527} C_VEL
LIN {X 0,Y 608.463,Z 630.551,A -85,B 0,C 180,E1 -531.531,E2 -531.531} C_VEL
LIN {X 0,Y 608.46,Z 638.838,A -85,B 0,C 180,E1 -532.701,E2 -532.701} C_VEL
LIN {X 0,Y 608.443,Z 645.325,A -85,B 0,C 180,E1 -533.831,E2 -533.831} C_VEL
LIN {X 0,Y 608.435,Z 650.787,A -85,B 0,C 180,E1 -535.03,E2 -535.03} C_VEL
LIN {X 0,Y 608.434,Z 654.297,A -85,B 0,C 180,E1 -536.026,E2 -536.026} C_VEL
LIN {X 0,Y 608.424,Z 657.734,A -85,B 0,C 180,E1 -537.352,E2 -537.352} C_VEL
LIN {X 0,Y 608.446,Z 659.778,A -85,B 0,C 180,E1 -538.676,E2 -538.676} C_VEL
LIN {X 0,Y 608.434,Z 660.495,A -85,B 0,C 180,E1 -540,E2 -540} C_VEL
LIN {X 0,Y 608.443,Z 659.881,A -85,B 0,C 180,E1 -541.324,E2 -541.324} C_VEL
LIN {X 0,Y 608.421,Z 657.928,A -85,B 0,C 180,E1 -542.648,E2 -542.648} C_VEL
LIN {X 0,Y 608.434,Z 654.585,A -85,B 0,C 180,E1 -543.974,E2 -543.974} C_VEL
LIN {X 0,Y 608.44,Z 649.76,A -85,B 0,C 180,E1 -545.302,E2 -545.302} C_VEL
LIN {X 0,Y 608.442,Z 643.433,A -85,B 0,C 180,E1 -546.608,E2 -546.608} C_VEL
LIN {X 0,Y 608.451,Z 636.1,A -85,B 0,C 180,E1 -547.8,E2 -547.8} C_VEL
LIN {X 0,Y 608.476,Z 628.56,A -85,B 0,C 180,E1 -548.803,E2 -548.803} C_VEL
LIN {X 0,Y 608.47,Z 626.658,A -85,B 0,C 180,E1 -549.033,E2 -549.033} C_VEL
LIN {X 0,Y 607.811,Z 622.971,A -85,B 0,C 180,E1 -549.46,E2 -549.46} C_VEL
LIN {X 0,Y 604.982,Z 616.737,A -85,B 0,C 180,E1 -550.142,E2 -550.142} C_VEL
LIN {X 0,Y 602.152,Z 610.165,A -85,B 0,C 180,E1 -550.794,E2 -550.794} C_VEL
LIN {X 0,Y 601.494,Z 605.791,A -85,B 0,C 180,E1 -551.169,E2 -551.169} C_VEL
LIN {X 0,Y 601.531,Z 594.814,A -85,B 0,C 180,E1 -551.969,E2 -551.969} C_VEL
LIN {X 0,Y 601.571,Z 581.905,A -85,B 0,C 180,E1 -552.739,E2 -552.739} C_VEL
LIN {X 0,Y 601.64,Z 568.218,A -85,B 0,C 180,E1 -553.382,E2 -553.382} C_VEL
LIN {X 0,Y 601.691,Z 553.909,A -85,B 0,C 180,E1 -553.886,E2 -553.886} C_VEL
LIN {X 0,Y 601.721,Z 539.295,A -85,B 0,C 180,E1 -554.244,E2 -554.244} C_VEL
LIN {X 0,Y 601.77,Z 520.884,A -85,B 0,C 180,E1 -554.508,E2 -554.508} C_VEL
LIN {X 0,Y 601.679,Z 398.345,A -85,B 0,C 180,E1 -555.997,E2 -555.997} C_VEL
LIN {X 0,Y 601.546,Z 397.014,A -85,B 0,C 180,E1 -556.066,E2 -556.066} C_VEL
LIN {X 0,Y 601.609,Z 373.797,A -85,B 0,C 180,E1 -558.872,E2 -558.872} C_VEL
LIN {X 0,Y 601.704,Z 351.707,A -85,B 0,C 180,E1 -561.588,E2 -561.588} C_VEL
LIN {X 0,Y 601.772,Z 332.874,A -85,B 0,C 180,E1 -563.944,E2 -563.944} C_VEL
LIN {X 0,Y 601.432,Z 330.339,A -85,B 0,C 180,E1 -564.317,E2 -564.317} C_VEL
LIN {X 0,Y 601.362,Z 330.196,A -85,B 0,C 180,E1 -567.116,E2 -567.116} C_VEL
LIN {X 0,Y 601.403,Z 330.2,A -85,B 0,C 180,E1 -570.165,E2 -570.165} C_VEL
LIN {X 0,Y 601.384,Z 330.194,A -85,B 0,C 180,E1 -572.71,E2 -572.71} C_VEL
LIN {X 0,Y 601.345,Z 330.198,A -85,B 0,C 180,E1 -575.105,E2 -575.105} C_VEL
LIN {X 0,Y 601.38,Z 330.195,A -85,B 0,C 180,E1 -577.423,E2 -577.423} C_VEL
LIN {X 0,Y 601.393,Z 330.202,A -85,B 0,C 180,E1 -579.997,E2 -579.997} C_VEL
LIN {X 0,Y 601.35,Z 330.198,A -85,B 0,C 180,E1 -582.676,E2 -582.676} C_VEL
LIN {X 0,Y 601.371,Z 330.198,A -85,B 0,C 180,E1 -584.53,E2 -584.53} C_VEL
LIN {X 0,Y 601.401,Z 330.194,A -85,B 0,C 180,E1 -586.43,E2 -586.43} C_VEL
LIN {X 0,Y 601.349,Z 330.197,A -85,B 0,C 180,E1 -589.12,E2 -589.12} C_VEL
LIN {X 0,Y 601.373,Z 330.199,A -85,B 0,C 180,E1 -591.728,E2 -591.728} C_VEL
LIN {X 0,Y 601.372,Z 330.202,A -85,B 0,C 180,E1 -594.244,E2 -594.244} C_VEL
LIN {X 0,Y 601.378,Z 330.195,A -85,B 0,C 180,E1 -596.683,E2 -596.683} C_VEL
LIN {X 0,Y 601.369,Z 330.195,A -85,B 0,C 180,E1 -599.055,E2 -599.055} C_VEL
LIN {X 0,Y 601.358,Z 330.198,A -85,B 0,C 180,E1 -601.369,E2 -601.369} C_VEL
LIN {X 0,Y 601.449,Z 330.416,A -85,B 0,C 180,E1 -603.768,E2 -603.768} C_VEL
LIN {X 0,Y 601.959,Z 333.691,A -85,B 0,C 180,E1 -604.179,E2 -604.179} C_VEL
LIN {X 0,Y 601.811,Z 355.254,A -85,B 0,C 180,E1 -606.606,E2 -606.606} C_VEL
LIN {X 0,Y 601.729,Z 380.287,A -85,B 0,C 180,E1 -609.373,E2 -609.373} C_VEL
LIN {X 0,Y 601.687,Z 398.665,A -85,B 0,C 180,E1 -611.354,E2 -611.354} C_VEL
LIN {X 0,Y 602.025,Z 402.637,A -85,B 0,C 180,E1 -611.429,E2 -611.429} C_VEL
LIN {X 0,Y 601.895,Z 564.61,A -85,B 0,C 180,E1 -613.429,E2 -613.429} C_VEL
LIN {X 0,Y 601.847,Z 579.769,A -85,B 0,C 180,E1 -613.746,E2 -613.746} C_VEL
LIN {X 0,Y 601.774,Z 594.765,A -85,B 0,C 180,E1 -614.201,E2 -614.201} C_VEL
LIN {X 0,Y 601.712,Z 608.732,A -85,B 0,C 180,E1 -614.764,E2 -614.764} C_VEL
LIN {X 0,Y 601.654,Z 622.409,A -85,B 0,C 180,E1 -615.455,E2 -615.455} C_VEL
LIN {X 0,Y 601.617,Z 635.792,A -85,B 0,C 180,E1 -616.283,E2 -616.283} C_VEL
LIN {X 0,Y 601.531,Z 647.729,A -85,B 0,C 180,E1 -617.174,E2 -617.174} C_VEL
LIN {X 0,Y 601.489,Z 659.271,A -85,B 0,C 180,E1 -618.201,E2 -618.201} C_VEL
LIN {X 0,Y 601.43,Z 668.998,A -85,B 0,C 180,E1 -619.224,E2 -619.224} C_VEL
LIN {X 0,Y 601.428,Z 678.53,A -85,B 0,C 180,E1 -620.414,E2 -620.414} C_VEL
LIN {X 0,Y 601.378,Z 686.456,A -85,B 0,C 180,E1 -621.6,E2 -621.6} C_VEL
LIN {X 0,Y 601.368,Z 693.873,A -85,B 0,C 180,E1 -622.951,E2 -622.951} C_VEL
LIN {X 0,Y 601.372,Z 699.762,A -85,B 0,C 180,E1 -624.299,E2 -624.299} C_VEL
LIN {X 0,Y 601.328,Z 703.243,A -85,B 0,C 180,E1 -625.307,E2 -625.307} C_VEL
LIN {X 0,Y 601.336,Z 706.793,A -85,B 0,C 180,E1 -626.65,E2 -626.65} C_VEL
LIN {X 0,Y 601.342,Z 709.137,A -85,B 0,C 180,E1 -627.991,E2 -627.991} C_VEL
LIN {X 0,Y 601.334,Z 710.33,A -85,B 0,C 180,E1 -629.33,E2 -629.33} C_VEL
LIN {X 0,Y 601.335,Z 710.361,A -85,B 0,C 180,E1 -630.67,E2 -630.67} C_VEL
LIN {X 0,Y 601.343,Z 709.242,A -85,B 0,C 180,E1 -632.009,E2 -632.009} C_VEL
LIN {X 0,Y 601.339,Z 706.985,A -85,B 0,C 180,E1 -633.35,E2 -633.35} C_VEL
LIN {X 0,Y 601.328,Z 703.527,A -85,B 0,C 180,E1 -634.693,E2 -634.693} C_VEL
LIN {X 0,Y 601.357,Z 698.794,A -85,B 0,C 180,E1 -636.038,E2 -636.038} C_VEL
LIN {X 0,Y 601.364,Z 692.662,A -85,B 0,C 180,E1 -637.386,E2 -637.386} C_VEL
LIN {X 0,Y 601.387,Z 684.953,A -85,B 0,C 180,E1 -638.738,E2 -638.738} C_VEL
LIN {X 0,Y 601.428,Z 676.71,A -85,B 0,C 180,E1 -639.925,E2 -639.925} C_VEL
LIN {X 0,Y 601.443,Z 666.352,A -85,B 0,C 180,E1 -641.164,E2 -641.164} C_VEL
LIN {X 0,Y 601.523,Z 654.791,A -85,B 0,C 180,E1 -642.311,E2 -642.311} C_VEL
LIN {X 0,Y 601.56,Z 642.296,A -85,B 0,C 180,E1 -643.34,E2 -643.34} C_VEL
LIN {X 0,Y 601.642,Z 629.773,A -85,B 0,C 180,E1 -644.2,E2 -644.2} C_VEL
LIN {X 0,Y 601.683,Z 616.034,A -85,B 0,C 180,E1 -644.977,E2 -644.977} C_VEL
LIN {X 0,Y 601.753,Z 601.707,A -85,B 0,C 180,E1 -645.626,E2 -645.626} C_VEL
LIN {X 0,Y 601.809,Z 587.577,A -85,B 0,C 180,E1 -646.124,E2 -646.124} C_VEL
LIN {X 0,Y 601.859,Z 572.868,A -85,B 0,C 180,E1 -646.506,E2 -646.506} C_VEL
LIN {X 0,Y 601.9,Z 557.028,A -85,B 0,C 180,E1 -646.771,E2 -646.771} C_VEL
LIN {X 0,Y 601.94,Z 400.3,A -85,B 0,C 180,E1 -648.693,E2 -648.693} C_VEL
LIN {X 0,Y 601.67,Z 398.41,A -85,B 0,C 180,E1 -648.753,E2 -648.753} C_VEL
LIN {X 0,Y 601.72,Z 374.007,A -85,B 0,C 180,E1 -651.407,E2 -651.407} C_VEL
LIN {X 0,Y 601.822,Z 352.798,A -85,B 0,C 180,E1 -653.759,E2 -653.759} C_VEL
LIN {X 0,Y 601.967,Z 333.123,A -85,B 0,C 180,E1 -655.976,E2 -655.976} C_VEL
LIN {X 0,Y 601.386,Z 330.277,A -85,B 0,C 180,E1 -656.365,E2 -656.365} C_VEL
LIN {X 0,Y 601.374,Z 330.197,A -85,B 0,C 180,E1 -659.395,E2 -659.395} C_VEL
LIN {X 0,Y 601.374,Z 330.201,A -85,B 0,C 180,E1 -661.729,E2 -661.729} C_VEL
LIN {X 0,Y 601.396,Z 330.199,A -85,B 0,C 180,E1 -664.12,E2 -664.12} C_VEL
LIN {X 0,Y 601.364,Z 330.197,A -85,B 0,C 180,E1 -666.586,E2 -666.586} C_VEL
LIN {X 0,Y 601.392,Z 330.196,A -85,B 0,C 180,E1 -669.53,E2 -669.53} C_VEL
LIN {X 0,Y 601.409,Z 330.199,A -85,B 0,C 180,E1 -671.766,E2 -671.766} C_VEL
LIN {X 0,Y 601.398,Z 330.192,A -85,B 0,C 180,E1 -674.532,E2 -674.532} C_VEL
LIN {X 0,Y 601.372,Z 330.198,A -85,B 0,C 180,E1 -677.413,E2 -677.413} C_VEL
LIN {X 0,Y 601.394,Z 330.199,A -85,B 0,C 180,E1 -680.003,E2 -680.003} C_VEL
LIN {X 0,Y 601.389,Z 330.193,A -85,B 0,C 180,E1 -682.624,E2 -682.624} C_VEL
LIN {X 0,Y 601.37,Z 330.195,A -85,B 0,C 180,E1 -685.065,E2 -685.065} C_VEL
LIN {X 0,Y 601.419,Z 330.195,A -85,B 0,C 180,E1 -687.483,E2 -687.483} C_VEL
LIN {X 0,Y 601.428,Z 330.196,A -85,B 0,C 180,E1 -689.852,E2 -689.852} C_VEL
LIN {X 0,Y 601.375,Z 330.193,A -85,B 0,C 180,E1 -692.645,E2 -692.645} C_VEL
LIN {X 0,Y 601.38,Z 330.196,A -85,B 0,C 180,E1 -695.12,E2 -695.12} C_VEL
LIN {X 0,Y 601.416,Z 330.195,A -85,B 0,C 180,E1 -697.395,E2 -697.395} C_VEL
LIN {X 0,Y 601.391,Z 330.194,A -85,B 0,C 180,E1 -700.19,E2 -700.19} C_VEL
LIN {X 0,Y 601.403,Z 330.192,A -85,B 0,C 180,E1 -703.013,E2 -703.013} C_VEL
LIN {X 0,Y 601.423,Z 330.193,A -85,B 0,C 180,E1 -705.908,E2 -705.908} C_VEL
LIN {X 0,Y 601.403,Z 330.19,A -85,B 0,C 180,E1 -708.541,E2 -708.541} C_VEL
LIN {X 0,Y 601.408,Z 330.196,A -85,B 0,C 180,E1 -711.262,E2 -711.262} C_VEL
LIN {X 0,Y 601.412,Z 330.192,A -85,B 0,C 180,E1 -713.963,E2 -713.963} C_VEL
LIN {X 0,Y 601.377,Z 330.194,A -85,B 0,C 180,E1 -716.65,E2 -716.65} C_VEL
LIN {X 0,Y 601.448,Z 330.194,A -85,B 0,C 180,E1 -719.33,E2 -719.33} C_VEL
LIN {X 0,Y 601.434,Z 330.188,A -85,B 0,C 180,E1 -722.009,E2 -722.009} C_VEL
LIN {X 0,Y 601.401,Z 330.192,A -85,B 0,C 180,E1 -724.692,E2 -724.692} C_VEL
LIN {X 0,Y 601.441,Z 330.195,A -85,B 0,C 180,E1 -727.385,E2 -727.385} C_VEL
LIN {X 0,Y 601.43,Z 330.188,A -85,B 0,C 180,E1 -730.095,E2 -730.095} C_VEL
LIN {X 0,Y 601.409,Z 330.193,A -85,B 0,C 180,E1 -732.828,E2 -732.828} C_VEL
LIN {X 0,Y 601.414,Z 330.194,A -85,B 0,C 180,E1 -735.591,E2 -735.591} C_VEL
LIN {X 0,Y 601.415,Z 330.189,A -85,B 0,C 180,E1 -738.392,E2 -738.392} C_VEL
LIN {X 0,Y 601.404,Z 330.201,A -85,B 0,C 180,E1 -741.239,E2 -741.239} C_VEL
LIN {X 0,Y 601.459,Z 330.183,A -85,B 0,C 180,E1 -744.14,E2 -744.14} C_VEL
LIN {X 0,Y 601.452,Z 330.194,A -85,B 0,C 180,E1 -747.111,E2 -747.111} C_VEL
LIN {X 0,Y 601.429,Z 330.187,A -85,B 0,C 180,E1 -750.149,E2 -750.149} C_VEL
LIN {X 0,Y 601.414,Z 330.193,A -85,B 0,C 180,E1 -752.714,E2 -752.714} C_VEL
LIN {X 0,Y 601.391,Z 330.203,A -85,B 0,C 180,E1 -755.111,E2 -755.111} C_VEL
LIN {X 0,Y 601.436,Z 330.191,A -85,B 0,C 180,E1 -757.419,E2 -757.419} C_VEL
LIN {X 0,Y 601.411,Z 330.188,A -85,B 0,C 180,E1 -759.995,E2 -759.995} C_VEL
LIN {X 0,Y 601.411,Z 330.194,A -85,B 0,C 180,E1 -762.67,E2 -762.67} C_VEL
LIN {X 0,Y 601.427,Z 330.189,A -85,B 0,C 180,E1 -765.482,E2 -765.482} C_VEL
LIN {X 0,Y 601.424,Z 330.19,A -85,B 0,C 180,E1 -768.407,E2 -768.407} C_VEL
LIN {X 0,Y 601.438,Z 330.196,A -85,B 0,C 180,E1 -770.876,E2 -770.876} C_VEL
LIN {X 0,Y 601.403,Z 330.193,A -85,B 0,C 180,E1 -773.417,E2 -773.417} C_VEL
LIN {X 0,Y 601.431,Z 330.188,A -85,B 0,C 180,E1 -776.065,E2 -776.065} C_VEL
LIN {X 0,Y 601.43,Z 330.195,A -85,B 0,C 180,E1 -779.059,E2 -779.059} C_VEL
LIN {X 0,Y 601.42,Z 330.191,A -85,B 0,C 180,E1 -781.373,E2 -781.373} C_VEL
LIN {X 0,Y 601.396,Z 330.195,A -85,B 0,C 180,E1 -783.636,E2 -783.636} C_VEL
LIN {X 0,Y 601.457,Z 330.366,A -85,B 0,C 180,E1 -784.5,E2 -784.5} C_VEL
LIN {X 0,Y 601.978,Z 332.621,A -85,B 0,C 180,E1 -784.778,E2 -784.778} C_VEL
LIN {X 0,Y 601.837,Z 360.18,A -85,B 0,C 180,E1 -787.572,E2 -787.572} C_VEL
LIN {X 0,Y 601.687,Z 390.209,A -85,B 0,C 180,E1 -790.556,E2 -790.556} C_VEL
LIN {X 0,Y 601.719,Z 398.11,A -85,B 0,C 180,E1 -791.309,E2 -791.309} C_VEL
LIN {X 0,Y 602.041,Z 401.959,A -85,B 0,C 180,E1 -791.376,E2 -791.376} C_VEL
LIN {X 0,Y 601.893,Z 565.202,A -85,B 0,C 180,E1 -793.392,E2 -793.392} C_VEL
LIN {X 0,Y 601.828,Z 580.713,A -85,B 0,C 180,E1 -793.724,E2 -793.724} C_VEL
LIN {X 0,Y 601.766,Z 596.05,A -85,B 0,C 180,E1 -794.201,E2 -794.201} C_VEL
LIN {X 0,Y 601.717,Z 609.761,A -85,B 0,C 180,E1 -794.764,E2 -794.764} C_VEL
LIN {X 0,Y 601.659,Z 623.234,A -85,B 0,C 180,E1 -795.455,E2 -795.455} C_VEL
LIN {X 0,Y 601.617,Z 636.45,A -85,B 0,C 180,E1 -796.283,E2 -796.283} C_VEL
LIN {X 0,Y 601.531,Z 648.285,A -85,B 0,C 180,E1 -797.174,E2 -797.174} C_VEL
LIN {X 0,Y 601.488,Z 659.749,A -85,B 0,C 180,E1 -798.201,E2 -798.201} C_VEL
LIN {X 0,Y 601.43,Z 669.389,A -85,B 0,C 180,E1 -799.224,E2 -799.224} C_VEL
LIN {X 0,Y 601.428,Z 678.855,A -85,B 0,C 180,E1 -800.415,E2 -800.415} C_VEL
LIN {X 0,Y 601.369,Z 686.73,A -85,B 0,C 180,E1 -801.6,E2 -801.6} C_VEL
LIN {X 0,Y 601.367,Z 694.088,A -85,B 0,C 180,E1 -802.952,E2 -802.952} C_VEL
LIN {X 0,Y 601.373,Z 699.924,A -85,B 0,C 180,E1 -804.299,E2 -804.299} C_VEL
LIN {X 0,Y 601.33,Z 703.383,A -85,B 0,C 180,E1 -805.307,E2 -805.307} C_VEL
LIN {X 0,Y 601.337,Z 706.886,A -85,B 0,C 180,E1 -806.65,E2 -806.65} C_VEL
LIN {X 0,Y 601.342,Z 709.192,A -85,B 0,C 180,E1 -807.991,E2 -807.991} C_VEL
LIN {X 0,Y 601.335,Z 710.35,A -85,B 0,C 180,E1 -809.33,E2 -809.33} C_VEL
LIN {X 0,Y 601.335,Z 710.35,A -85,B 0,C 180,E1 -810.67,E2 -810.67} C_VEL
LIN {X 0,Y 601.342,Z 709.192,A -85,B 0,C 180,E1 -812.009,E2 -812.009} C_VEL
LIN {X 0,Y 601.337,Z 706.885,A -85,B 0,C 180,E1 -813.35,E2 -813.35} C_VEL
LIN {X 0,Y 601.33,Z 703.383,A -85,B 0,C 180,E1 -814.693,E2 -814.693} C_VEL
LIN {X 0,Y 601.356,Z 698.607,A -85,B 0,C 180,E1 -816.038,E2 -816.038} C_VEL
LIN {X 0,Y 601.365,Z 692.425,A -85,B 0,C 180,E1 -817.386,E2 -817.386} C_VEL
LIN {X 0,Y 601.386,Z 684.652,A -85,B 0,C 180,E1 -818.738,E2 -818.738} C_VEL
LIN {X 0,Y 601.428,Z 676.369,A -85,B 0,C 180,E1 -819.925,E2 -819.925} C_VEL
LIN {X 0,Y 601.46,Z 665.932,A -85,B 0,C 180,E1 -821.165,E2 -821.165} C_VEL
LIN {X 0,Y 601.515,Z 656.191,A -85,B 0,C 180,E1 -822.141,E2 -822.141} C_VEL
LIN {X 0,Y 601.57,Z 644.014,A -85,B 0,C 180,E1 -823.169,E2 -823.169} C_VEL
LIN {X 0,Y 601.607,Z 632.075,A -85,B 0,C 180,E1 -824.012,E2 -824.012} C_VEL
LIN {X 0,Y 601.665,Z 618.524,A -85,B 0,C 180,E1 -824.805,E2 -824.805} C_VEL
LIN {X 0,Y 601.761,Z 603.839,A -85,B 0,C 180,E1 -825.495,E2 -825.495} C_VEL
LIN {X 0,Y 601.785,Z 589.614,A -85,B 0,C 180,E1 -826.016,E2 -826.016} C_VEL
LIN {X 0,Y 601.864,Z 574.581,A -85,B 0,C 180,E1 -826.422,E2 -826.422} C_VEL
LIN {X 0,Y 601.878,Z 559.483,A -85,B 0,C 180,E1 -826.693,E2 -826.693} C_VEL
LIN {X 0,Y 601.955,Z 399.679,A -85,B 0,C 180,E1 -828.655,E2 -828.655} C_VEL
LIN {X 0,Y 601.699,Z 397.718,A -85,B 0,C 180,E1 -828.72,E2 -828.72} C_VEL
LIN {X 0,Y 601.747,Z 370.411,A -85,B 0,C 180,E1 -831.406,E2 -831.406} C_VEL
LIN {X 0,Y 601.93,Z 343.417,A -85,B 0,C 180,E1 -834.12,E2 -834.12} C_VEL
LIN {X 0,Y 601.98,Z 332.619,A -85,B 0,C 180,E1 -835.222,E2 -835.222} C_VEL
LIN {X 0,Y 601.433,Z 330.287,A -85,B 0,C 180,E1 -835.525,E2 -835.525} C_VEL
LIN {X 0,Y 601.402,Z 330.193,A -85,B 0,C 180,E1 -837.868,E2 -837.868} C_VEL
LIN {X 0,Y 601.43,Z 330.188,A -85,B 0,C 180,E1 -840.164,E2 -840.164} C_VEL
LIN {X 0,Y 601.417,Z 330.195,A -85,B 0,C 180,E1 -842.715,E2 -842.715} C_VEL
LIN {X 0,Y 601.398,Z 330.199,A -85,B 0,C 180,E1 -845.112,E2 -845.112} C_VEL
LIN {X 0,Y 601.434,Z 330.189,A -85,B 0,C 180,E1 -847.419,E2 -847.419} C_VEL
LIN {X 0,Y 601.402,Z 330.192,A -85,B 0,C 180,E1 -849.996,E2 -849.996} C_VEL
LIN {X 0,Y 601.409,Z 330.201,A -85,B 0,C 180,E1 -852.671,E2 -852.671} C_VEL
LIN {X 0,Y 601.399,Z 330.192,A -85,B 0,C 180,E1 -855.48,E2 -855.48} C_VEL
LIN {X 0,Y 601.423,Z 330.197,A -85,B 0,C 180,E1 -858.407,E2 -858.407} C_VEL
LIN {X 0,Y 601.392,Z 330.196,A -85,B 0,C 180,E1 -860.872,E2 -860.872} C_VEL
LIN {X 0,Y 601.382,Z 330.194,A -85,B 0,C 180,E1 -863.416,E2 -863.416} C_VEL
LIN {X 0,Y 601.429,Z 330.194,A -85,B 0,C 180,E1 -866.065,E2 -866.065} C_VEL
LIN {X 0,Y 601.387,Z 330.194,A -85,B 0,C 180,E1 -869.056,E2 -869.056} C_VEL
LIN {X 0,Y 601.366,Z 330.197,A -85,B 0,C 180,E1 -871.37,E2 -871.37} C_VEL
LIN {X 0,Y 601.392,Z 330.201,A -85,B 0,C 180,E1 -874.381,E2 -874.381} C_VEL
LIN {X 0,Y 601.425,Z 330.391,A -85,B 0,C 180,E1 -875.789,E2 -875.789} C_VEL
LIN {X 0,Y 601.77,Z 333.611,A -85,B 0,C 180,E1 -876.239,E2 -876.239} C_VEL
LIN {X 0,Y 601.687,Z 353.879,A -85,B 0,C 180,E1 -878.771,E2 -878.771} C_VEL
LIN {X 0,Y 601.597,Z 375.558,A -85,B 0,C 180,E1 -881.433,E2 -881.433} C_VEL
LIN {X 0,Y 601.578,Z 397.526,A -85,B 0,C 180,E1 -884.065,E2 -884.065} C_VEL
LIN {X 0,Y 601.859,Z 403.283,A -85,B 0,C 180,E1 -884.16,E2 -884.16} C_VEL
LIN {X 0,Y 601.732,Z 535.04,A -85,B 0,C 180,E1 -885.767,E2 -885.767} C_VEL
LIN {X 0,Y 601.712,Z 549.537,A -85,B 0,C 180,E1 -886.081,E2 -886.081} C_VEL
LIN {X 0,Y 601.668,Z 563.666,A -85,B 0,C 180,E1 -886.533,E2 -886.533} C_VEL
LIN {X 0,Y 601.6,Z 576.713,A -85,B 0,C 180,E1 -887.09,E2 -887.09} C_VEL
LIN {X 0,Y 601.551,Z 589.359,A -85,B 0,C 180,E1 -887.775,E2 -887.775} C_VEL
LIN {X 0,Y 601.505,Z 600.852,A -85,B 0,C 180,E1 -888.543,E2 -888.543} C_VEL
LIN {X 0,Y 601.481,Z 611.425,A -85,B 0,C 180,E1 -889.395,E2 -889.395} C_VEL
LIN {X 0,Y 601.431,Z 621.904,A -85,B 0,C 180,E1 -890.415,E2 -890.415} C_VEL
LIN {X 0,Y 601.406,Z 630.556,A -85,B 0,C 180,E1 -891.431,E2 -891.431} C_VEL
LIN {X 0,Y 601.391,Z 638.835,A -85,B 0,C 180,E1 -892.614,E2 -892.614} C_VEL
LIN {X 0,Y 601.361,Z 644.508,A -85,B 0,C 180,E1 -893.605,E2 -893.605} C_VEL
LIN {X 0,Y 601.354,Z 649.382,A -85,B 0,C 180,E1 -894.635,E2 -894.635} C_VEL
LIN {X 0,Y 601.345,Z 654.298,A -85,B 0,C 180,E1 -895.979,E2 -895.979} C_VEL
LIN {X 0,Y 601.324,Z 657.738,A -85,B 0,C 180,E1 -897.321,E2 -897.321} C_VEL
LIN {X 0,Y 601.345,Z 659.779,A -85,B 0,C 180,E1 -898.661,E2 -898.661} C_VEL
LIN {X 0,Y 601.334,Z 660.496,A -85,B 0,C 180,E1 -900,E2 -900} C_VEL
LIN {X 0,Y 601.342,Z 659.876,A -85,B 0,C 180,E1 -901.339,E2 -901.339} C_VEL
LIN {X 0,Y 601.321,Z 657.929,A -85,B 0,C 180,E1 -902.68,E2 -902.68} C_VEL
LIN {X 0,Y 601.346,Z 654.583,A -85,B 0,C 180,E1 -904.021,E2 -904.021} C_VEL
LIN {X 0,Y 601.355,Z 649.761,A -85,B 0,C 180,E1 -905.365,E2 -905.365} C_VEL
LIN {X 0,Y 601.368,Z 643.886,A -85,B 0,C 180,E1 -906.601,E2 -906.601} C_VEL
LIN {X 0,Y 601.384,Z 637.221,A -85,B 0,C 180,E1 -907.724,E2 -907.724} C_VEL
LIN {X 0,Y 601.411,Z 628.553,A -85,B 0,C 180,E1 -908.907,E2 -908.907} C_VEL
LIN {X 0,Y 601.431,Z 619.517,A -85,B 0,C 180,E1 -909.925,E2 -909.925} C_VEL
LIN {X 0,Y 601.475,Z 608.329,A -85,B 0,C 180,E1 -910.964,E2 -910.964} C_VEL
LIN {X 0,Y 601.494,Z 605.791,A -85,B 0,C 180,E1 -911.169,E2 -911.169} C_VEL
LIN {X 0,Y 600.838,Z 601.3,A -85,B 0,C 180,E1 -911.53,E2 -911.53} C_VEL
LIN {X 0,Y 598.029,Z 593.925,A -85,B 0,C 180,E1 -912.106,E2 -912.106} C_VEL
LIN {X 0,Y 595.25,Z 586.2,A -85,B 0,C 180,E1 -912.639,E2 -912.639} C_VEL
LIN {X 0,Y 594.635,Z 581.165,A -85,B 0,C 180,E1 -912.929,E2 -912.929} C_VEL
LIN {X 0,Y 594.732,Z 568.204,A -85,B 0,C 180,E1 -913.54,E2 -913.54} C_VEL
LIN {X 0,Y 594.79,Z 554.556,A -85,B 0,C 180,E1 -914.03,E2 -914.03} C_VEL
LIN {X 0,Y 594.849,Z 540.517,A -85,B 0,C 180,E1 -914.388,E2 -914.388} C_VEL
LIN {X 0,Y 594.882,Z 525.133,A -85,B 0,C 180,E1 -914.627,E2 -914.627} C_VEL
LIN {X 0,Y 594.977,Z 399.897,A -85,B 0,C 180,E1 -916.16,E2 -916.16} C_VEL
LIN {X 0,Y 594.568,Z 397.235,A -85,B 0,C 180,E1 -916.238,E2 -916.238} C_VEL
LIN {X 0,Y 594.672,Z 373.752,A -85,B 0,C 180,E1 -919.105,E2 -919.105} C_VEL
LIN {X 0,Y 594.835,Z 350.253,A -85,B 0,C 180,E1 -922.032,E2 -922.032} C_VEL
LIN {X 0,Y 594.918,Z 334.318,A -85,B 0,C 180,E1 -924.052,E2 -924.052} C_VEL
LIN {X 0,Y 594.385,Z 331.204,A -85,B 0,C 180,E1 -924.516,E2 -924.516} C_VEL
LIN {X 0,Y 594.326,Z 331.076,A -85,B 0,C 180,E1 -927.515,E2 -927.515} C_VEL
LIN {X 0,Y 594.364,Z 331.074,A -85,B 0,C 180,E1 -930.324,E2 -930.324} C_VEL
LIN {X 0,Y 594.335,Z 331.071,A -85,B 0,C 180,E1 -932.953,E2 -932.953} C_VEL
LIN {X 0,Y 594.302,Z 331.077,A -85,B 0,C 180,E1 -935.412,E2 -935.412} C_VEL
LIN {X 0,Y 594.346,Z 331.079,A -85,B 0,C 180,E1 -937.944,E2 -937.944} C_VEL
LIN {X 0,Y 594.322,Z 331.073,A -85,B 0,C 180,E1 -940.816,E2 -940.816} C_VEL
LIN {X 0,Y 594.334,Z 331.071,A -85,B 0,C 180,E1 -943.303,E2 -943.303} C_VEL
LIN {X 0,Y 594.333,Z 331.079,A -85,B 0,C 180,E1 -946.164,E2 -946.164} C_VEL
LIN {X 0,Y 594.35,Z 331.072,A -85,B 0,C 180,E1 -948.533,E2 -948.533} C_VEL
LIN {X 0,Y 594.324,Z 331.073,A -85,B 0,C 180,E1 -951.303,E2 -951.303} C_VEL
LIN {X 0,Y 594.338,Z 331.076,A -85,B 0,C 180,E1 -953.754,E2 -953.754} C_VEL
LIN {X 0,Y 594.341,Z 331.078,A -85,B 0,C 180,E1 -956.236,E2 -956.236} C_VEL
LIN {X 0,Y 594.322,Z 331.075,A -85,B 0,C 180,E1 -958.647,E2 -958.647} C_VEL
LIN {X 0,Y 594.331,Z 331.073,A -85,B 0,C 180,E1 -961.052,E2 -961.052} C_VEL
LIN {X 0,Y 594.36,Z 331.212,A -85,B 0,C 180,E1 -963.512,E2 -963.512} C_VEL
LIN {X 0,Y 595.173,Z 335.695,A -85,B 0,C 180,E1 -964.093,E2 -964.093} C_VEL
LIN {X 0,Y 594.979,Z 358.521,A -85,B 0,C 180,E1 -966.69,E2 -966.69} C_VEL
LIN {X 0,Y 594.844,Z 384.607,A -85,B 0,C 180,E1 -969.602,E2 -969.602} C_VEL
LIN {X 0,Y 594.778,Z 398.667,A -85,B 0,C 180,E1 -971.128,E2 -971.128} C_VEL
LIN {X 0,Y 595.3,Z 402.744,A -85,B 0,C 180,E1 -971.212,E2 -971.212} C_VEL
LIN {X 0,Y 595.098,Z 564.715,A -85,B 0,C 180,E1 -973.236,E2 -973.236} C_VEL
LIN {X 0,Y 595.023,Z 580.678,A -85,B 0,C 180,E1 -973.576,E2 -973.576} C_VEL
LIN {X 0,Y 594.916,Z 595.963,A -85,B 0,C 180,E1 -974.058,E2 -974.058} C_VEL
LIN {X 0,Y 594.833,Z 608.742,A -85,B 0,C 180,E1 -974.583,E2 -974.583} C_VEL
LIN {X 0,Y 594.737,Z 622.418,A -85,B 0,C 180,E1 -975.282,E2 -975.282} C_VEL
LIN {X 0,Y 594.682,Z 635.144,A -85,B 0,C 180,E1 -976.075,E2 -976.075} C_VEL
LIN {X 0,Y 594.56,Z 647.737,A -85,B 0,C 180,E1 -977.021,E2 -977.021} C_VEL
LIN {X 0,Y 594.467,Z 659.271,A -85,B 0,C 180,E1 -978.06,E2 -978.06} C_VEL
LIN {X 0,Y 594.39,Z 669.006,A -85,B 0,C 180,E1 -979.095,E2 -979.095} C_VEL
LIN {X 0,Y 594.381,Z 678.537,A -85,B 0,C 180,E1 -980.3,E2 -980.3} C_VEL
LIN {X 0,Y 594.318,Z 686.457,A -85,B 0,C 180,E1 -981.499,E2 -981.499} C_VEL
LIN {X 0,Y 594.292,Z 693.878,A -85,B 0,C 180,E1 -982.867,E2 -982.867} C_VEL
LIN {X 0,Y 594.297,Z 699.767,A -85,B 0,C 180,E1 -984.231,E2 -984.231} C_VEL
LIN {X 0,Y 594.23,Z 703.246,A -85,B 0,C 180,E1 -985.251,E2 -985.251} C_VEL
LIN {X 0,Y 594.256,Z 706.797,A -85,B 0,C 180,E1 -986.61,E2 -986.61} C_VEL
LIN {X 0,Y 594.241,Z 709.136,A -85,B 0,C 180,E1 -987.967,E2 -987.967} C_VEL
LIN {X 0,Y 594.235,Z 710.323,A -85,B 0,C 180,E1 -989.322,E2 -989.322} C_VEL
LIN {X 0,Y 594.236,Z 710.356,A -85,B 0,C 180,E1 -990.678,E2 -990.678} C_VEL
LIN {X 0,Y 594.241,Z 709.24,A -85,B 0,C 180,E1 -992.033,E2 -992.033} C_VEL
LIN {X 0,Y 594.259,Z 706.987,A -85,B 0,C 180,E1 -993.39,E2 -993.39} C_VEL
LIN {X 0,Y 594.231,Z 703.527,A -85,B 0,C 180,E1 -994.749,E2 -994.749} C_VEL
LIN {X 0,Y 594.278,Z 698.786,A -85,B 0,C 180,E1 -996.11,E2 -996.11} C_VEL
LIN {X 0,Y 594.287,Z 692.652,A -85,B 0,C 180,E1 -997.474,E2 -997.474} C_VEL
LIN {X 0,Y 594.331,Z 684.951,A -85,B 0,C 180,E1 -998.843,E2 -998.843} C_VEL
LIN {X 0,Y 594.388,Z 676.706,A -85,B 0,C 180,E1 -1000.044,E2 -1000.044} C_VEL
LIN {X 0,Y 594.411,Z 666.96,A -85,B 0,C 180,E1 -1001.229,E2 -1001.229} C_VEL
LIN {X 0,Y 594.514,Z 656.638,A -85,B 0,C 180,E1 -1002.286,E2 -1002.286} C_VEL
LIN {X 0,Y 594.579,Z 644.593,A -85,B 0,C 180,E1 -1003.326,E2 -1003.326} C_VEL
LIN {X 0,Y 594.687,Z 631.076,A -85,B 0,C 180,E1 -1004.286,E2 -1004.286} C_VEL
LIN {X 0,Y 594.774,Z 617.716,A -85,B 0,C 180,E1 -1005.067,E2 -1005.067} C_VEL
LIN {X 0,Y 594.883,Z 602.813,A -85,B 0,C 180,E1 -1005.767,E2 -1005.767} C_VEL
LIN {X 0,Y 594.98,Z 588.257,A -85,B 0,C 180,E1 -1006.292,E2 -1006.292} C_VEL
LIN {X 0,Y 595.043,Z 573.55,A -85,B 0,C 180,E1 -1006.684,E2 -1006.684} C_VEL
LIN {X 0,Y 595.112,Z 557.667,A -85,B 0,C 180,E1 -1006.96,E2 -1006.96} C_VEL
LIN {X 0,Y 595.209,Z 401.201,A -85,B 0,C 180,E1 -1008.901,E2 -1008.901} C_VEL
LIN {X 0,Y 594.741,Z 398.314,A -85,B 0,C 180,E1 -1008.987,E2 -1008.987} C_VEL
LIN {X 0,Y 594.871,Z 374.002,A -85,B 0,C 180,E1 -1011.666,E2 -1011.666} C_VEL
LIN {X 0,Y 595.082,Z 349.53,A -85,B 0,C 180,E1 -1014.416,E2 -1014.416} C_VEL
LIN {X 0,Y 595.075,Z 334.341,A -85,B 0,C 180,E1 -1016.158,E2 -1016.158} C_VEL
LIN {X 0,Y 594.344,Z 331.215,A -85,B 0,C 180,E1 -1016.578,E2 -1016.578} C_VEL
LIN {X 0,Y 594.347,Z 331.078,A -85,B 0,C 180,E1 -1019.778,E2 -1019.778} C_VEL
LIN {X 0,Y 594.336,Z 331.079,A -85,B 0,C 180,E1 -1022.149,E2 -1022.149} C_VEL
LIN {X 0,Y 594.339,Z 331.073,A -85,B 0,C 180,E1 -1024.583,E2 -1024.583} C_VEL
LIN {X 0,Y 594.349,Z 331.075,A -85,B 0,C 180,E1 -1027.603,E2 -1027.603} C_VEL
LIN {X 0,Y 594.323,Z 331.074,A -85,B 0,C 180,E1 -1030.571,E2 -1030.571} C_VEL
LIN {X 0,Y 594.314,Z 331.074,A -85,B 0,C 180,E1 -1032.847,E2 -1032.847} C_VEL
LIN {X 0,Y 594.337,Z 331.072,A -85,B 0,C 180,E1 -1035.194,E2 -1035.194} C_VEL
LIN {X 0,Y 594.373,Z 331.071,A -85,B 0,C 180,E1 -1038.153,E2 -1038.153} C_VEL
LIN {X 0,Y 594.361,Z 331.07,A -85,B 0,C 180,E1 -1041.298,E2 -1041.298} C_VEL
LIN {X 0,Y 594.343,Z 331.08,A -85,B 0,C 180,E1 -1043.755,E2 -1043.755} C_VEL
LIN {X 0,Y 594.359,Z 331.071,A -85,B 0,C 180,E1 -1046.237,E2 -1046.237} C_VEL
LIN {X 0,Y 594.358,Z 331.068,A -85,B 0,C 180,E1 -1048.649,E2 -1048.649} C_VEL
LIN {X 0,Y 594.374,Z 331.068,A -85,B 0,C 180,E1 -1051.044,E2 -1051.044} C_VEL
LIN {X 0,Y 594.357,Z 331.072,A -85,B 0,C 180,E1 -1054.055,E2 -1054.055} C_VEL
LIN {X 0,Y 594.37,Z 331.068,A -85,B 0,C 180,E1 -1056.295,E2 -1056.295} C_VEL
LIN {X 0,Y 594.395,Z 331.067,A -85,B 0,C 180,E1 -1059.224,E2 -1059.224} C_VEL
LIN {X 0,Y 594.341,Z 331.072,A -85,B 0,C 180,E1 -1062.095,E2 -1062.095} C_VEL
LIN {X 0,Y 594.353,Z 331.07,A -85,B 0,C 180,E1 -1064.219,E2 -1064.219} C_VEL
LIN {X 0,Y 594.37,Z 331.067,A -85,B 0,C 180,E1 -1066.321,E2 -1066.321} C_VEL
LIN {X 0,Y 594.352,Z 331.071,A -85,B 0,C 180,E1 -1069.094,E2 -1069.094} C_VEL
LIN {X 0,Y 594.411,Z 331.066,A -85,B 0,C 180,E1 -1071.843,E2 -1071.843} C_VEL
LIN {X 0,Y 594.371,Z 331.066,A -85,B 0,C 180,E1 -1074.572,E2 -1074.572} C_VEL
LIN {X 0,Y 594.406,Z 331.069,A -85,B 0,C 180,E1 -1077.289,E2 -1077.289} C_VEL
LIN {X 0,Y 594.414,Z 331.062,A -85,B 0,C 180,E1 -1080,E2 -1080} C_VEL
LIN {X 0,Y 594.388,Z 331.065,A -85,B 0,C 180,E1 -1082.711,E2 -1082.711} C_VEL
LIN {X 0,Y 594.397,Z 331.072,A -85,B 0,C 180,E1 -1085.428,E2 -1085.428} C_VEL
LIN {X 0,Y 594.383,Z 331.064,A -85,B 0,C 180,E1 -1088.157,E2 -1088.157} C_VEL
LIN {X 0,Y 594.38,Z 331.072,A -85,B 0,C 180,E1 -1091.068,E2 -1091.068} C_VEL
LIN {X 0,Y 594.385,Z 331.068,A -85,B 0,C 180,E1 -1093.679,E2 -1093.679} C_VEL
LIN {X 0,Y 594.368,Z 331.069,A -85,B 0,C 180,E1 -1096.71,E2 -1096.71} C_VEL
LIN {X 0,Y 594.368,Z 331.075,A -85,B 0,C 180,E1 -1099.334,E2 -1099.334} C_VEL
LIN {X 0,Y 594.364,Z 331.073,A -85,B 0,C 180,E1 -1101.503,E2 -1101.503} C_VEL
LIN {X 0,Y 594.39,Z 331.064,A -85,B 0,C 180,E1 -1104.446,E2 -1104.446} C_VEL
LIN {X 0,Y 594.383,Z 331.068,A -85,B 0,C 180,E1 -1106.7,E2 -1106.7} C_VEL
LIN {X 0,Y 594.38,Z 331.074,A -85,B 0,C 180,E1 -1108.998,E2 -1108.998} C_VEL
LIN {X 0,Y 594.383,Z 331.068,A -85,B 0,C 180,E1 -1111.644,E2 -1111.644} C_VEL
LIN {X 0,Y 594.377,Z 331.068,A -85,B 0,C 180,E1 -1114.58,E2 -1114.58} C_VEL
LIN {X 0,Y 594.391,Z 331.066,A -85,B 0,C 180,E1 -1117.609,E2 -1117.609} C_VEL
LIN {X 0,Y 594.37,Z 331.067,A -85,B 0,C 180,E1 -1120.567,E2 -1120.567} C_VEL
LIN {X 0,Y 594.367,Z 331.073,A -85,B 0,C 180,E1 -1123.299,E2 -1123.299} C_VEL
LIN {X 0,Y 594.368,Z 331.066,A -85,B 0,C 180,E1 -1126.16,E2 -1126.16} C_VEL
LIN {X 0,Y 594.381,Z 331.068,A -85,B 0,C 180,E1 -1128.536,E2 -1128.536} C_VEL
LIN {X 0,Y 594.388,Z 331.069,A -85,B 0,C 180,E1 -1131.295,E2 -1131.295} C_VEL
LIN {X 0,Y 594.352,Z 331.069,A -85,B 0,C 180,E1 -1133.756,E2 -1133.756} C_VEL
LIN {X 0,Y 594.377,Z 331.068,A -85,B 0,C 180,E1 -1136.239,E2 -1136.239} C_VEL
LIN {X 0,Y 594.39,Z 331.071,A -85,B 0,C 180,E1 -1138.651,E2 -1138.651} C_VEL
LIN {X 0,Y 594.381,Z 331.072,A -85,B 0,C 180,E1 -1141.043,E2 -1141.043} C_VEL
LIN {X 0,Y 594.382,Z 331.071,A -85,B 0,C 180,E1 -1143.978,E2 -1143.978} C_VEL
LIN {X 0,Y 594.432,Z 331.373,A -85,B 0,C 180,E1 -1144.294,E2 -1144.294} C_VEL
LIN {X 0,Y 595.172,Z 334.421,A -85,B 0,C 180,E1 -1144.656,E2 -1144.656} C_VEL
LIN {X 0,Y 595.042,Z 356.016,A -85,B 0,C 180,E1 -1146.877,E2 -1146.877} C_VEL
LIN {X 0,Y 594.861,Z 383.01,A -85,B 0,C 180,E1 -1149.603,E2 -1149.603} C_VEL
LIN {X 0,Y 594.808,Z 398.041,A -85,B 0,C 180,E1 -1151.08,E2 -1151.08} C_VEL
LIN {X 0,Y 595.317,Z 401.808,A -85,B 0,C 180,E1 -1151.156,E2 -1151.156} C_VEL
LIN {X 0,Y 595.104,Z 564.93,A -85,B 0,C 180,E1 -1153.192,E2 -1153.192} C_VEL
LIN {X 0,Y 595.007,Z 580.712,A -85,B 0,C 180,E1 -1153.532,E2 -1153.532} C_VEL
LIN {X 0,Y 594.933,Z 596.048,A -85,B 0,C 180,E1 -1154.015,E2 -1154.015} C_VEL
LIN {X 0,Y 594.856,Z 609.763,A -85,B 0,C 180,E1 -1154.584,E2 -1154.584} C_VEL
LIN {X 0,Y 594.735,Z 623.237,A -85,B 0,C 180,E1 -1155.282,E2 -1155.282} C_VEL
LIN {X 0,Y 594.68,Z 635.793,A -85,B 0,C 180,E1 -1156.075,E2 -1156.075} C_VEL
LIN {X 0,Y 594.559,Z 648.286,A -85,B 0,C 180,E1 -1157.021,E2 -1157.021} C_VEL
LIN {X 0,Y 594.466,Z 659.749,A -85,B 0,C 180,E1 -1158.06,E2 -1158.06} C_VEL
LIN {X 0,Y 594.388,Z 669.39,A -85,B 0,C 180,E1 -1159.095,E2 -1159.095} C_VEL
LIN {X 0,Y 594.367,Z 678.856,A -85,B 0,C 180,E1 -1160.3,E2 -1160.3} C_VEL
LIN {X 0,Y 594.311,Z 686.731,A -85,B 0,C 180,E1 -1161.5,E2 -1161.5} C_VEL
LIN {X 0,Y 594.291,Z 694.088,A -85,B 0,C 180,E1 -1162.867,E2 -1162.867} C_VEL
LIN {X 0,Y 594.298,Z 699.924,A -85,B 0,C 180,E1 -1164.231,E2 -1164.231} C_VEL
LIN {X 0,Y 594.232,Z 703.384,A -85,B 0,C 180,E1 -1165.251,E2 -1165.251} C_VEL
LIN {X 0,Y 594.257,Z 706.887,A -85,B 0,C 180,E1 -1166.61,E2 -1166.61} C_VEL
LIN {X 0,Y 594.241,Z 709.193,A -85,B 0,C 180,E1 -1167.967,E2 -1167.967} C_VEL
LIN {X 0,Y 594.235,Z 710.35,A -85,B 0,C 180,E1 -1169.322,E2 -1169.322} C_VEL
LIN {X 0,Y 594.235,Z 710.35,A -85,B 0,C 180,E1 -1170.678,E2 -1170.678} C_VEL
LIN {X 0,Y 594.241,Z 709.192,A -85,B 0,C 180,E1 -1172.033,E2 -1172.033} C_VEL
LIN {X 0,Y 594.257,Z 706.886,A -85,B 0,C 180,E1 -1173.39,E2 -1173.39} C_VEL
LIN {X 0,Y 594.232,Z 703.383,A -85,B 0,C 180,E1 -1174.749,E2 -1174.749} C_VEL
LIN {X 0,Y 594.278,Z 698.607,A -85,B 0,C 180,E1 -1176.11,E2 -1176.11} C_VEL
LIN {X 0,Y 594.287,Z 692.424,A -85,B 0,C 180,E1 -1177.475,E2 -1177.475} C_VEL
LIN {X 0,Y 594.33,Z 684.651,A -85,B 0,C 180,E1 -1178.843,E2 -1178.843} C_VEL
LIN {X 0,Y 594.388,Z 676.369,A -85,B 0,C 180,E1 -1180.044,E2 -1180.044} C_VEL
LIN {X 0,Y 594.433,Z 666.559,A -85,B 0,C 180,E1 -1181.231,E2 -1181.231} C_VEL
LIN {X 0,Y 594.531,Z 656.19,A -85,B 0,C 180,E1 -1182.285,E2 -1182.285} C_VEL
LIN {X 0,Y 594.581,Z 644.015,A -85,B 0,C 180,E1 -1183.326,E2 -1183.326} C_VEL
LIN {X 0,Y 594.695,Z 632.073,A -85,B 0,C 180,E1 -1184.178,E2 -1184.178} C_VEL
LIN {X 0,Y 594.763,Z 618.522,A -85,B 0,C 180,E1 -1184.98,E2 -1184.98} C_VEL
LIN {X 0,Y 594.901,Z 603.837,A -85,B 0,C 180,E1 -1185.679,E2 -1185.679} C_VEL
LIN {X 0,Y 594.955,Z 589.613,A -85,B 0,C 180,E1 -1186.205,E2 -1186.205} C_VEL
LIN {X 0,Y 595.054,Z 575.033,A -85,B 0,C 180,E1 -1186.605,E2 -1186.605} C_VEL
LIN {X 0,Y 595.077,Z 559.483,A -85,B 0,C 180,E1 -1186.889,E2 -1186.889} C_VEL
LIN {X 0,Y 595.191,Z 400.264,A -85,B 0,C 180,E1 -1188.868,E2 -1188.868} C_VEL
LIN {X 0,Y 594.812,Z 397.82,A -85,B 0,C 180,E1 -1188.936,E2 -1188.936} C_VEL
LIN {X 0,Y 594.957,Z 368.612,A -85,B 0,C 180,E1 -1191.845,E2 -1191.845} C_VEL
LIN {X 0,Y 595.184,Z 341.574,A -85,B 0,C 180,E1 -1194.602,E2 -1194.602} C_VEL
LIN {X 0,Y 595.172,Z 334.419,A -85,B 0,C 180,E1 -1195.344,E2 -1195.344} C_VEL
LIN {X 0,Y 594.394,Z 331.169,A -85,B 0,C 180,E1 -1195.755,E2 -1195.755} C_VEL
LIN {X 0,Y 594.372,Z 331.069,A -85,B 0,C 180,E1 -1198.227,E2 -1198.227} C_VEL
LIN {X 0,Y 594.382,Z 331.069,A -85,B 0,C 180,E1 -1200.56,E2 -1200.56} C_VEL
LIN {X 0,Y 594.377,Z 331.076,A -85,B 0,C 180,E1 -1202.95,E2 -1202.95} C_VEL
LIN {X 0,Y 594.354,Z 331.072,A -85,B 0,C 180,E1 -1205.409,E2 -1205.409} C_VEL
LIN {X 0,Y 594.388,Z 331.066,A -85,B 0,C 180,E1 -1207.941,E2 -1207.941} C_VEL
LIN {X 0,Y 594.374,Z 331.076,A -85,B 0,C 180,E1 -1210.822,E2 -1210.822} C_VEL
LIN {X 0,Y 594.352,Z 331.071,A -85,B 0,C 180,E1 -1213.301,E2 -1213.301} C_VEL
LIN {X 0,Y 594.361,Z 331.072,A -85,B 0,C 180,E1 -1216.161,E2 -1216.161} C_VEL
LIN {X 0,Y 594.379,Z 331.076,A -85,B 0,C 180,E1 -1218.536,E2 -1218.536} C_VEL
LIN {X 0,Y 594.367,Z 331.068,A -85,B 0,C 180,E1 -1221.298,E2 -1221.298} C_VEL
LIN {X 0,Y 594.346,Z 331.072,A -85,B 0,C 180,E1 -1223.755,E2 -1223.755} C_VEL
LIN {X 0,Y 594.371,Z 331.077,A -85,B 0,C 180,E1 -1226.238,E2 -1226.238} C_VEL
LIN {X 0,Y 594.358,Z 331.073,A -85,B 0,C 180,E1 -1228.649,E2 -1228.649} C_VEL
LIN {X 0,Y 594.335,Z 331.073,A -85,B 0,C 180,E1 -1231.051,E2 -1231.051} C_VEL
LIN {X 0,Y 594.35,Z 331.079,A -85,B 0,C 180,E1 -1233.985,E2 -1233.985} C_VEL
LIN {X 0,Y 594.378,Z 331.289,A -85,B 0,C 180,E1 -1235.6,E2 -1235.6} C_VEL
LIN {X 0,Y 594.919,Z 335.063,A -85,B 0,C 180,E1 -1236.134,E2 -1236.134} C_VEL
LIN {X 0,Y 594.788,Z 355.075,A -85,B 0,C 180,E1 -1238.662,E2 -1238.662} C_VEL
LIN {X 0,Y 594.668,Z 375.915,A -85,B 0,C 180,E1 -1241.252,E2 -1241.252} C_VEL
LIN {X 0,Y 594.618,Z 397.536,A -85,B 0,C 180,E1 -1243.874,E2 -1243.874} C_VEL
LIN {X 0,Y 595.002,Z 401.54,A -85,B 0,C 180,E1 -1243.951,E2 -1243.951} C_VEL
LIN {X 0,Y 594.865,Z 535.849,A -85,B 0,C 180,E1 -1245.613,E2 -1245.613} C_VEL
LIN {X 0,Y 594.806,Z 550.318,A -85,B 0,C 180,E1 -1245.937,E2 -1245.937} C_VEL
LIN {X 0,Y 594.754,Z 564.806,A -85,B 0,C 180,E1 -1246.417,E2 -1246.417} C_VEL
LIN {X 0,Y 594.638,Z 578.473,A -85,B 0,C 180,E1 -1247.023,E2 -1247.023} C_VEL
LIN {X 0,Y 594.595,Z 590.785,A -85,B 0,C 180,E1 -1247.716,E2 -1247.716} C_VEL
LIN {X 0,Y 594.528,Z 603.033,A -85,B 0,C 180,E1 -1248.569,E2 -1248.569} C_VEL
LIN {X 0,Y 594.448,Z 613.352,A -85,B 0,C 180,E1 -1249.441,E2 -1249.441} C_VEL
LIN {X 0,Y 594.372,Z 623.47,A -85,B 0,C 180,E1 -1250.472,E2 -1250.472} C_VEL
LIN {X 0,Y 594.324,Z 631.842,A -85,B 0,C 180,E1 -1251.5,E2 -1251.5} C_VEL
LIN {X 0,Y 594.303,Z 639.865,A -85,B 0,C 180,E1 -1252.697,E2 -1252.697} C_VEL
LIN {X 0,Y 594.28,Z 646.317,A -85,B 0,C 180,E1 -1253.89,E2 -1253.89} C_VEL
LIN {X 0,Y 594.245,Z 650.781,A -85,B 0,C 180,E1 -1254.911,E2 -1254.911} C_VEL
LIN {X 0,Y 594.261,Z 654.299,A -85,B 0,C 180,E1 -1255.931,E2 -1255.931} C_VEL
LIN {X 0,Y 594.224,Z 657.741,A -85,B 0,C 180,E1 -1257.288,E2 -1257.288} C_VEL
LIN {X 0,Y 594.245,Z 659.78,A -85,B 0,C 180,E1 -1258.645,E2 -1258.645} C_VEL
LIN {X 0,Y 594.235,Z 660.496,A -85,B 0,C 180,E1 -1260,E2 -1260} C_VEL
LIN {X 0,Y 594.242,Z 659.87,A -85,B 0,C 180,E1 -1261.355,E2 -1261.355} C_VEL
LIN {X 0,Y 594.222,Z 657.929,A -85,B 0,C 180,E1 -1262.712,E2 -1262.712} C_VEL
LIN {X 0,Y 594.262,Z 654.582,A -85,B 0,C 180,E1 -1264.069,E2 -1264.069} C_VEL
LIN {X 0,Y 594.275,Z 649.762,A -85,B 0,C 180,E1 -1265.429,E2 -1265.429} C_VEL
LIN {X 0,Y 594.277,Z 644.376,A -85,B 0,C 180,E1 -1266.587,E2 -1266.587} C_VEL
LIN {X 0,Y 594.315,Z 637.221,A -85,B 0,C 180,E1 -1267.816,E2 -1267.816} C_VEL
LIN {X 0,Y 594.368,Z 628.546,A -85,B 0,C 180,E1 -1269.014,E2 -1269.014} C_VEL
LIN {X 0,Y 594.4,Z 619.515,A -85,B 0,C 180,E1 -1270.044,E2 -1270.044} C_VEL
LIN {X 0,Y 594.478,Z 609.208,A -85,B 0,C 180,E1 -1271.017,E2 -1271.017} C_VEL
LIN {X 0,Y 594.572,Z 597.359,A -85,B 0,C 180,E1 -1271.938,E2 -1271.938} C_VEL
LIN {X 0,Y 594.613,Z 585.034,A -85,B 0,C 180,E1 -1272.717,E2 -1272.717} C_VEL
LIN {X 0,Y 594.635,Z 581.165,A -85,B 0,C 180,E1 -1272.929,E2 -1272.929} C_VEL
LIN {X 0,Y 593.981,Z 577.746,A -85,B 0,C 180,E1 -1273.12,E2 -1273.12} C_VEL
LIN {X 0,Y 588.453,Z 567.132,A -85,B 0,C 180,E1 -1273.731,E2 -1273.731} C_VEL
LIN {X 0,Y 587.859,Z 563.544,A -85,B 0,C 180,E1 -1273.885,E2 -1273.885} C_VEL
LIN {X 0,Y 587.912,Z 549.333,A -85,B 0,C 180,E1 -1274.348,E2 -1274.348} C_VEL
LIN {X 0,Y 588,Z 534.604,A -85,B 0,C 180,E1 -1274.669,E2 -1274.669} C_VEL
LIN {X 0,Y 588.086,Z 400.41,A -85,B 0,C 180,E1 -1276.348,E2 -1276.348} C_VEL
LIN {X 0,Y 587.642,Z 397.56,A -85,B 0,C 180,E1 -1276.412,E2 -1276.412} C_VEL
LIN {X 0,Y 587.721,Z 375.301,A -85,B 0,C 180,E1 -1279.145,E2 -1279.145} C_VEL
LIN {X 0,Y 587.923,Z 354.594,A -85,B 0,C 180,E1 -1281.751,E2 -1281.751} C_VEL
LIN {X 0,Y 588.073,Z 335.938,A -85,B 0,C 180,E1 -1284.139,E2 -1284.139} C_VEL
LIN {X 0,Y 587.331,Z 332.096,A -85,B 0,C 180,E1 -1284.711,E2 -1284.711} C_VEL
LIN {X 0,Y 587.285,Z 331.955,A -85,B 0,C 180,E1 -1287.68,E2 -1287.68} C_VEL
LIN {X 0,Y 587.308,Z 331.95,A -85,B 0,C 180,E1 -1290.505,E2 -1290.505} C_VEL
LIN {X 0,Y 587.303,Z 331.949,A -85,B 0,C 180,E1 -1293.399,E2 -1293.399} C_VEL
LIN {X 0,Y 587.268,Z 331.96,A -85,B 0,C 180,E1 -1295.902,E2 -1295.902} C_VEL
LIN {X 0,Y 587.281,Z 331.953,A -85,B 0,C 180,E1 -1298.483,E2 -1298.483} C_VEL
LIN {X 0,Y 587.282,Z 331.949,A -85,B 0,C 180,E1 -1301.162,E2 -1301.162} C_VEL
LIN {X 0,Y 587.288,Z 331.959,A -85,B 0,C 180,E1 -1304.109,E2 -1304.109} C_VEL
LIN {X 0,Y 587.27,Z 331.95,A -85,B 0,C 180,E1 -1306.989,E2 -1306.989} C_VEL
LIN {X 0,Y 587.286,Z 331.959,A -85,B 0,C 180,E1 -1309.986,E2 -1309.986} C_VEL
LIN {X 0,Y 587.301,Z 331.952,A -85,B 0,C 180,E1 -1312.389,E2 -1312.389} C_VEL
LIN {X 0,Y 587.316,Z 331.95,A -85,B 0,C 180,E1 -1315.657,E2 -1315.657} C_VEL
LIN {X 0,Y 587.299,Z 331.956,A -85,B 0,C 180,E1 -1318.228,E2 -1318.228} C_VEL
LIN {X 0,Y 587.295,Z 331.951,A -85,B 0,C 180,E1 -1320.876,E2 -1320.876} C_VEL
LIN {X 0,Y 587.324,Z 332.162,A -85,B 0,C 180,E1 -1323.29,E2 -1323.29} C_VEL
LIN {X 0,Y 588.403,Z 337.331,A -85,B 0,C 180,E1 -1323.963,E2 -1323.963} C_VEL
LIN {X 0,Y 588.187,Z 358.526,A -85,B 0,C 180,E1 -1326.404,E2 -1326.404} C_VEL
LIN {X 0,Y 587.977,Z 384.613,A -85,B 0,C 180,E1 -1329.353,E2 -1329.353} C_VEL
LIN {X 0,Y 587.856,Z 398.808,A -85,B 0,C 180,E1 -1330.904,E2 -1330.904} C_VEL
LIN {X 0,Y 588.591,Z 402.633,A -85,B 0,C 180,E1 -1330.987,E2 -1330.987} C_VEL
LIN {X 0,Y 588.291,Z 564.384,A -85,B 0,C 180,E1 -1333.031,E2 -1333.031} C_VEL
LIN {X 0,Y 588.224,Z 579.813,A -85,B 0,C 180,E1 -1333.359,E2 -1333.359} C_VEL
LIN {X 0,Y 588.085,Z 594.799,A -85,B 0,C 180,E1 -1333.823,E2 -1333.823} C_VEL
LIN {X 0,Y 587.97,Z 608.737,A -85,B 0,C 180,E1 -1334.399,E2 -1334.399} C_VEL
LIN {X 0,Y 587.837,Z 622.427,A -85,B 0,C 180,E1 -1335.105,E2 -1335.105} C_VEL
LIN {X 0,Y 587.748,Z 635.508,A -85,B 0,C 180,E1 -1335.932,E2 -1335.932} C_VEL
LIN {X 0,Y 587.582,Z 647.746,A -85,B 0,C 180,E1 -1336.864,E2 -1336.864} C_VEL
LIN {X 0,Y 587.455,Z 659.272,A -85,B 0,C 180,E1 -1337.915,E2 -1337.915} C_VEL
LIN {X 0,Y 587.351,Z 669.014,A -85,B 0,C 180,E1 -1338.963,E2 -1338.963} C_VEL
LIN {X 0,Y 587.31,Z 678.545,A -85,B 0,C 180,E1 -1340.182,E2 -1340.182} C_VEL
LIN {X 0,Y 587.268,Z 686.458,A -85,B 0,C 180,E1 -1341.397,E2 -1341.397} C_VEL
LIN {X 0,Y 587.216,Z 693.882,A -85,B 0,C 180,E1 -1342.781,E2 -1342.781} C_VEL
LIN {X 0,Y 587.226,Z 699.772,A -85,B 0,C 180,E1 -1344.161,E2 -1344.161} C_VEL
LIN {X 0,Y 587.134,Z 703.249,A -85,B 0,C 180,E1 -1345.193,E2 -1345.193} C_VEL
LIN {X 0,Y 587.179,Z 706.801,A -85,B 0,C 180,E1 -1346.569,E2 -1346.569} C_VEL
LIN {X 0,Y 587.139,Z 709.136,A -85,B 0,C 180,E1 -1347.942,E2 -1347.942} C_VEL
LIN {X 0,Y 587.135,Z 710.317,A -85,B 0,C 180,E1 -1349.314,E2 -1349.314} C_VEL
LIN {X 0,Y 587.136,Z 710.349,A -85,B 0,C 180,E1 -1350.686,E2 -1350.686} C_VEL
LIN {X 0,Y 587.14,Z 709.238,A -85,B 0,C 180,E1 -1352.058,E2 -1352.058} C_VEL
LIN {X 0,Y 587.181,Z 706.989,A -85,B 0,C 180,E1 -1353.431,E2 -1353.431} C_VEL
LIN {X 0,Y 587.134,Z 703.527,A -85,B 0,C 180,E1 -1354.806,E2 -1354.806} C_VEL
LIN {X 0,Y 587.182,Z 698.778,A -85,B 0,C 180,E1 -1356.184,E2 -1356.184} C_VEL
LIN {X 0,Y 587.229,Z 692.642,A -85,B 0,C 180,E1 -1357.565,E2 -1357.565} C_VEL
LIN {X 0,Y 587.266,Z 684.948,A -85,B 0,C 180,E1 -1358.95,E2 -1358.95} C_VEL
LIN {X 0,Y 587.352,Z 676.7,A -85,B 0,C 180,E1 -1360.165,E2 -1360.165} C_VEL
LIN {X 0,Y 587.377,Z 666.762,A -85,B 0,C 180,E1 -1361.386,E2 -1361.386} C_VEL
LIN {X 0,Y 587.513,Z 656.625,A -85,B 0,C 180,E1 -1362.434,E2 -1362.434} C_VEL
LIN {X 0,Y 587.62,Z 644.586,A -85,B 0,C 180,E1 -1363.487,E2 -1363.487} C_VEL
LIN {X 0,Y 587.762,Z 631.786,A -85,B 0,C 180,E1 -1364.411,E2 -1364.411} C_VEL
LIN {X 0,Y 587.872,Z 619.294,A -85,B 0,C 180,E1 -1365.16,E2 -1365.16} C_VEL
LIN {X 0,Y 587.999,Z 606.819,A -85,B 0,C 180,E1 -1365.778,E2 -1365.778} C_VEL
LIN {X 0,Y 588.118,Z 592.265,A -85,B 0,C 180,E1 -1366.354,E2 -1366.354} C_VEL
LIN {X 0,Y 588.248,Z 577.229,A -85,B 0,C 180,E1 -1366.794,E2 -1366.794} C_VEL
LIN {X 0,Y 588.316,Z 562.443,A -85,B 0,C 180,E1 -1367.09,E2 -1367.09} C_VEL
LIN {X 0,Y 588.523,Z 402.22,A -85,B 0,C 180,E1 -1369.11,E2 -1369.11} C_VEL
LIN {X 0,Y 587.846,Z 398.384,A -85,B 0,C 180,E1 -1369.212,E2 -1369.212} C_VEL
LIN {X 0,Y 588.043,Z 372.365,A -85,B 0,C 180,E1 -1372.115,E2 -1372.115} C_VEL
LIN {X 0,Y 588.332,Z 346.588,A -85,B 0,C 180,E1 -1375.054,E2 -1375.054} C_VEL
LIN {X 0,Y 588.337,Z 336.472,A -85,B 0,C 180,E1 -1376.231,E2 -1376.231} C_VEL
LIN {X 0,Y 587.315,Z 332.053,A -85,B 0,C 180,E1 -1376.83,E2 -1376.83} C_VEL
LIN {X 0,Y 587.293,Z 331.953,A -85,B 0,C 180,E1 -1379.382,E2 -1379.382} C_VEL
LIN {X 0,Y 587.293,Z 331.956,A -85,B 0,C 180,E1 -1381.827,E2 -1381.827} C_VEL
LIN {X 0,Y 587.316,Z 331.95,A -85,B 0,C 180,E1 -1384.343,E2 -1384.343} C_VEL
LIN {X 0,Y 587.304,Z 331.952,A -85,B 0,C 180,E1 -1387.611,E2 -1387.611} C_VEL
LIN {X 0,Y 587.285,Z 331.954,A -85,B 0,C 180,E1 -1390.257,E2 -1390.257} C_VEL
LIN {X 0,Y 587.277,Z 331.951,A -85,B 0,C 180,E1 -1393.114,E2 -1393.114} C_VEL
LIN {X 0,Y 587.298,Z 331.955,A -85,B 0,C 180,E1 -1396.047,E2 -1396.047} C_VEL
LIN {X 0,Y 587.285,Z 331.95,A -85,B 0,C 180,E1 -1398.931,E2 -1398.931} C_VEL
LIN {X 0,Y 587.31,Z 331.952,A -85,B 0,C 180,E1 -1401.519,E2 -1401.519} C_VEL
LIN {X 0,Y 587.275,Z 331.955,A -85,B 0,C 180,E1 -1404.099,E2 -1404.099} C_VEL
LIN {X 0,Y 587.333,Z 331.944,A -85,B 0,C 180,E1 -1406.889,E2 -1406.889} C_VEL
LIN {X 0,Y 587.328,Z 331.952,A -85,B 0,C 180,E1 -1409.829,E2 -1409.829} C_VEL
LIN {X 0,Y 587.301,Z 331.948,A -85,B 0,C 180,E1 -1412.317,E2 -1412.317} C_VEL
LIN {X 0,Y 587.351,Z 331.947,A -85,B 0,C 180,E1 -1415.42,E2 -1415.42} C_VEL
LIN {X 0,Y 587.314,Z 331.947,A -85,B 0,C 180,E1 -1418.225,E2 -1418.225} C_VEL
LIN {X 0,Y 587.336,Z 331.946,A -85,B 0,C 180,E1 -1421.151,E2 -1421.151} C_VEL
LIN {X 0,Y 587.31,Z 331.949,A -85,B 0,C 180,E1 -1424.024,E2 -1424.024} C_VEL
LIN {X 0,Y 587.352,Z 331.943,A -85,B 0,C 180,E1 -1426.154,E2 -1426.154} C_VEL
LIN {X 0,Y 587.338,Z 331.943,A -85,B 0,C 180,E1 -1428.962,E2 -1428.962} C_VEL
LIN {X 0,Y 587.363,Z 331.946,A -85,B 0,C 180,E1 -1431.745,E2 -1431.745} C_VEL
LIN {X 0,Y 587.339,Z 331.941,A -85,B 0,C 180,E1 -1434.507,E2 -1434.507} C_VEL
LIN {X 0,Y 587.37,Z 331.945,A -85,B 0,C 180,E1 -1437.257,E2 -1437.257} C_VEL
LIN {X 0,Y 587.383,Z 331.938,A -85,B 0,C 180,E1 -1440,E2 -1440} C_VEL
LIN {X 0,Y 587.357,Z 331.94,A -85,B 0,C 180,E1 -1442.743,E2 -1442.743} C_VEL
LIN {X 0,Y 587.363,Z 331.947,A -85,B 0,C 180,E1 -1445.493,E2 -1445.493} C_VEL
LIN {X 0,Y 587.342,Z 331.941,A -85,B 0,C 180,E1 -1448.256,E2 -1448.256} C_VEL
LIN {X 0,Y 587.35,Z 331.948,A -85,B 0,C 180,E1 -1451.134,E2 -1451.134} C_VEL
LIN {X 0,Y 587.342,Z 331.941,A -85,B 0,C 180,E1 -1454.251,E2 -1454.251} C_VEL
LIN {X 0,Y 587.346,Z 331.949,A -85,B 0,C 180,E1 -1457.406,E2 -1457.406} C_VEL
LIN {X 0,Y 587.324,Z 331.943,A -85,B 0,C 180,E1 -1460.305,E2 -1460.305} C_VEL
LIN {X 0,Y 587.316,Z 331.954,A -85,B 0,C 180,E1 -1463.259,E2 -1463.259} C_VEL
LIN {X 0,Y 587.332,Z 331.948,A -85,B 0,C 180,E1 -1465.517,E2 -1465.517} C_VEL
LIN {X 0,Y 587.346,Z 331.943,A -85,B 0,C 180,E1 -1467.818,E2 -1467.818} C_VEL
LIN {X 0,Y 587.339,Z 331.943,A -85,B 0,C 180,E1 -1470.51,E2 -1470.51} C_VEL
LIN {X 0,Y 587.334,Z 331.948,A -85,B 0,C 180,E1 -1473.397,E2 -1473.397} C_VEL
LIN {X 0,Y 587.292,Z 331.949,A -85,B 0,C 180,E1 -1475.9,E2 -1475.9} C_VEL
LIN {X 0,Y 587.334,Z 331.945,A -85,B 0,C 180,E1 -1478.479,E2 -1478.479} C_VEL
LIN {X 0,Y 587.337,Z 331.95,A -85,B 0,C 180,E1 -1481.157,E2 -1481.157} C_VEL
LIN {X 0,Y 587.327,Z 331.944,A -85,B 0,C 180,E1 -1484.113,E2 -1484.113} C_VEL
LIN {X 0,Y 587.314,Z 331.953,A -85,B 0,C 180,E1 -1486.994,E2 -1486.994} C_VEL
LIN {X 0,Y 587.319,Z 331.946,A -85,B 0,C 180,E1 -1489.746,E2 -1489.746} C_VEL
LIN {X 0,Y 587.346,Z 331.945,A -85,B 0,C 180,E1 -1492.392,E2 -1492.392} C_VEL
LIN {X 0,Y 587.359,Z 331.941,A -85,B 0,C 180,E1 -1495.78,E2 -1495.78} C_VEL
LIN {X 0,Y 587.35,Z 331.943,A -85,B 0,C 180,E1 -1498.232,E2 -1498.232} C_VEL
LIN {X 0,Y 587.348,Z 331.952,A -85,B 0,C 180,E1 -1500.867,E2 -1500.867} C_VEL
LIN {X 0,Y 587.358,Z 331.948,A -85,B 0,C 180,E1 -1503.819,E2 -1503.819} C_VEL
LIN {X 0,Y 587.38,Z 332.323,A -85,B 0,C 180,E1 -1504.066,E2 -1504.066} C_VEL
LIN {X 0,Y 588.391,Z 336.22,A -85,B 0,C 180,E1 -1504.533,E2 -1504.533} C_VEL
LIN {X 0,Y 588.24,Z 357.816,A -85,B 0,C 180,E1 -1506.78,E2 -1506.78} C_VEL
LIN {X 0,Y 588.006,Z 384.81,A -85,B 0,C 180,E1 -1509.537,E2 -1509.537} C_VEL
LIN {X 0,Y 587.905,Z 397.901,A -85,B 0,C 180,E1 -1510.84,E2 -1510.84} C_VEL
LIN {X 0,Y 588.623,Z 402.949,A -85,B 0,C 180,E1 -1510.947,E2 -1510.947} C_VEL
LIN {X 0,Y 588.321,Z 564.956,A -85,B 0,C 180,E1 -1512.993,E2 -1512.993} C_VEL
LIN {X 0,Y 588.203,Z 580.711,A -85,B 0,C 180,E1 -1513.336,E2 -1513.336} C_VEL
LIN {X 0,Y 588.07,Z 596.046,A -85,B 0,C 180,E1 -1513.823,E2 -1513.823} C_VEL
LIN {X 0,Y 587.987,Z 609.766,A -85,B 0,C 180,E1 -1514.399,E2 -1514.399} C_VEL
LIN {X 0,Y 587.833,Z 623.239,A -85,B 0,C 180,E1 -1515.105,E2 -1515.105} C_VEL
LIN {X 0,Y 587.74,Z 636.114,A -85,B 0,C 180,E1 -1515.929,E2 -1515.929} C_VEL
LIN {X 0,Y 587.582,Z 648.288,A -85,B 0,C 180,E1 -1516.864,E2 -1516.864} C_VEL
LIN {X 0,Y 587.454,Z 659.749,A -85,B 0,C 180,E1 -1517.915,E2 -1517.915} C_VEL
LIN {X 0,Y 587.348,Z 669.391,A -85,B 0,C 180,E1 -1518.963,E2 -1518.963} C_VEL
LIN {X 0,Y 587.305,Z 678.857,A -85,B 0,C 180,E1 -1520.182,E2 -1520.182} C_VEL
LIN {X 0,Y 587.264,Z 686.732,A -85,B 0,C 180,E1 -1521.397,E2 -1521.397} C_VEL
LIN {X 0,Y 587.215,Z 694.089,A -85,B 0,C 180,E1 -1522.781,E2 -1522.781} C_VEL
LIN {X 0,Y 587.226,Z 699.924,A -85,B 0,C 180,E1 -1524.161,E2 -1524.161} C_VEL
LIN {X 0,Y 587.136,Z 703.384,A -85,B 0,C 180,E1 -1525.194,E2 -1525.194} C_VEL
LIN {X 0,Y 587.18,Z 706.888,A -85,B 0,C 180,E1 -1526.569,E2 -1526.569} C_VEL
LIN {X 0,Y 587.14,Z 709.193,A -85,B 0,C 180,E1 -1527.942,E2 -1527.942} C_VEL
LIN {X 0,Y 587.135,Z 710.35,A -85,B 0,C 180,E1 -1529.314,E2 -1529.314} C_VEL
LIN {X 0,Y 587.135,Z 710.349,A -85,B 0,C 180,E1 -1530.686,E2 -1530.686} C_VEL
LIN {X 0,Y 587.14,Z 709.193,A -85,B 0,C 180,E1 -1532.058,E2 -1532.058} C_VEL
LIN {X 0,Y 587.18,Z 706.886,A -85,B 0,C 180,E1 -1533.431,E2 -1533.431} C_VEL
LIN {X 0,Y 587.136,Z 703.384,A -85,B 0,C 180,E1 -1534.807,E2 -1534.807} C_VEL
LIN {X 0,Y 587.179,Z 698.608,A -85,B 0,C 180,E1 -1536.184,E2 -1536.184} C_VEL
LIN {X 0,Y 587.23,Z 692.424,A -85,B 0,C 180,E1 -1537.565,E2 -1537.565} C_VEL
LIN {X 0,Y 587.265,Z 684.65,A -85,B 0,C 180,E1 -1538.95,E2 -1538.95} C_VEL
LIN {X 0,Y 587.352,Z 676.369,A -85,B 0,C 180,E1 -1540.166,E2 -1540.166} C_VEL
LIN {X 0,Y 587.4,Z 666.394,A -85,B 0,C 180,E1 -1541.386,E2 -1541.386} C_VEL
LIN {X 0,Y 587.522,Z 656.189,A -85,B 0,C 180,E1 -1542.434,E2 -1542.434} C_VEL
LIN {X 0,Y 587.629,Z 644.016,A -85,B 0,C 180,E1 -1543.487,E2 -1543.487} C_VEL
LIN {X 0,Y 587.775,Z 631.054,A -85,B 0,C 180,E1 -1544.416,E2 -1544.416} C_VEL
LIN {X 0,Y 587.886,Z 616.863,A -85,B 0,C 180,E1 -1545.248,E2 -1545.248} C_VEL
LIN {X 0,Y 588.048,Z 602.792,A -85,B 0,C 180,E1 -1545.911,E2 -1545.911} C_VEL
LIN {X 0,Y 588.169,Z 588.299,A -85,B 0,C 180,E1 -1546.442,E2 -1546.442} C_VEL
LIN {X 0,Y 588.289,Z 573.193,A -85,B 0,C 180,E1 -1546.846,E2 -1546.846} C_VEL
LIN {X 0,Y 588.326,Z 557.958,A -85,B 0,C 180,E1 -1547.112,E2 -1547.112} C_VEL
LIN {X 0,Y 588.569,Z 401.658,A -85,B 0,C 180,E1 -1549.071,E2 -1549.071} C_VEL
LIN {X 0,Y 587.921,Z 397.897,A -85,B 0,C 180,E1 -1549.16,E2 -1549.16} C_VEL
LIN {X 0,Y 588.082,Z 372.211,A -85,B 0,C 180,E1 -1551.745,E2 -1551.745} C_VEL
LIN {X 0,Y 588.375,Z 345.217,A -85,B 0,C 180,E1 -1554.525,E2 -1554.525} C_VEL
LIN {X 0,Y 588.39,Z 336.219,A -85,B 0,C 180,E1 -1555.468,E2 -1555.468} C_VEL
LIN {X 0,Y 587.358,Z 332.068,A -85,B 0,C 180,E1 -1555.988,E2 -1555.988} C_VEL
LIN {X 0,Y 587.32,Z 331.951,A -85,B 0,C 180,E1 -1558.597,E2 -1558.597} C_VEL
LIN {X 0,Y 587.33,Z 331.954,A -85,B 0,C 180,E1 -1560.967,E2 -1560.967} C_VEL
LIN {X 0,Y 587.334,Z 331.948,A -85,B 0,C 180,E1 -1563.397,E2 -1563.397} C_VEL
LIN {X 0,Y 587.299,Z 331.949,A -85,B 0,C 180,E1 -1565.9,E2 -1565.9} C_VEL
LIN {X 0,Y 587.33,Z 331.949,A -85,B 0,C 180,E1 -1568.48,E2 -1568.48} C_VEL
LIN {X 0,Y 587.334,Z 331.948,A -85,B 0,C 180,E1 -1571.157,E2 -1571.157} C_VEL
LIN {X 0,Y 587.319,Z 331.948,A -85,B 0,C 180,E1 -1574.113,E2 -1574.113} C_VEL
LIN {X 0,Y 587.298,Z 331.952,A -85,B 0,C 180,E1 -1576.992,E2 -1576.992} C_VEL
LIN {X 0,Y 587.307,Z 331.948,A -85,B 0,C 180,E1 -1579.745,E2 -1579.745} C_VEL
LIN {X 0,Y 587.34,Z 331.953,A -85,B 0,C 180,E1 -1582.392,E2 -1582.392} C_VEL
LIN {X 0,Y 587.349,Z 331.945,A -85,B 0,C 180,E1 -1585.779,E2 -1585.779} C_VEL
LIN {X 0,Y 587.332,Z 331.954,A -85,B 0,C 180,E1 -1588.231,E2 -1588.231} C_VEL
LIN {X 0,Y 587.299,Z 331.951,A -85,B 0,C 180,E1 -1590.876,E2 -1590.876} C_VEL
LIN {X 0,Y 587.302,Z 331.956,A -85,B 0,C 180,E1 -1593.831,E2 -1593.831} C_VEL
LIN {X 0,Y 587.311,Z 332.08,A -85,B 0,C 180,E1 -1595.371,E2 -1595.371} C_VEL
LIN {X 0,Y 587.999,Z 335.25,A -85,B 0,C 180,E1 -1595.858,E2 -1595.858} C_VEL
LIN {X 0,Y 587.95,Z 350.993,A -85,B 0,C 180,E1 -1597.881,E2 -1597.881} C_VEL
LIN {X 0,Y 587.745,Z 373.403,A -85,B 0,C 180,E1 -1600.708,E2 -1600.708} C_VEL
LIN {X 0,Y 587.6,Z 395.876,A -85,B 0,C 180,E1 -1603.497,E2 -1603.497} C_VEL
LIN {X 0,Y 587.661,Z 397.839,A -85,B 0,C 180,E1 -1603.689,E2 -1603.689} C_VEL
LIN {X 0,Y 588.206,Z 401.586,A -85,B 0,C 180,E1 -1603.76,E2 -1603.76} C_VEL
LIN {X 0,Y 587.997,Z 535.887,A -85,B 0,C 180,E1 -1605.441,E2 -1605.441} C_VEL
LIN {X 0,Y 587.926,Z 550.598,A -85,B 0,C 180,E1 -1605.776,E2 -1605.776} C_VEL
LIN {X 0,Y 587.853,Z 564.824,A -85,B 0,C 180,E1 -1606.254,E2 -1606.254} C_VEL
LIN {X 0,Y 587.7,Z 578.481,A -85,B 0,C 180,E1 -1606.867,E2 -1606.867} C_VEL
LIN {X 0,Y 587.617,Z 590.799,A -85,B 0,C 180,E1 -1607.568,E2 -1607.568} C_VEL
LIN {X 0,Y 587.514,Z 602.022,A -85,B 0,C 180,E1 -1608.354,E2 -1608.354} C_VEL
LIN {X 0,Y 587.444,Z 613.351,A -85,B 0,C 180,E1 -1609.313,E2 -1609.313} C_VEL
LIN {X 0,Y 587.324,Z 623.477,A -85,B 0,C 180,E1 -1610.356,E2 -1610.356} C_VEL
LIN {X 0,Y 587.278,Z 633.082,A -85,B 0,C 180,E1 -1611.57,E2 -1611.57} C_VEL
LIN {X 0,Y 587.226,Z 640.881,A -85,B 0,C 180,E1 -1612.781,E2 -1612.781} C_VEL
LIN {X 0,Y 587.203,Z 646.321,A -85,B 0,C 180,E1 -1613.816,E2 -1613.816} C_VEL
LIN {X 0,Y 587.158,Z 650.778,A -85,B 0,C 180,E1 -1614.85,E2 -1614.85} C_VEL
LIN {X 0,Y 587.181,Z 654.299,A -85,B 0,C 180,E1 -1615.882,E2 -1615.882} C_VEL
LIN {X 0,Y 587.13,Z 657.745,A -85,B 0,C 180,E1 -1617.256,E2 -1617.256} C_VEL
LIN {X 0,Y 587.145,Z 659.776,A -85,B 0,C 180,E1 -1618.628,E2 -1618.628} C_VEL
LIN {X 0,Y 587.136,Z 660.496,A -85,B 0,C 180,E1 -1620,E2 -1620} C_VEL
LIN {X 0,Y 587.142,Z 659.864,A -85,B 0,C 180,E1 -1621.372,E2 -1621.372} C_VEL
LIN {X 0,Y 587.128,Z 657.929,A -85,B 0,C 180,E1 -1622.744,E2 -1622.744} C_VEL
LIN {X 0,Y 587.181,Z 654.577,A -85,B 0,C 180,E1 -1624.118,E2 -1624.118} C_VEL
LIN {X 0,Y 587.2,Z 649.762,A -85,B 0,C 180,E1 -1625.495,E2 -1625.495} C_VEL
LIN {X 0,Y 587.209,Z 644.754,A -85,B 0,C 180,E1 -1626.593,E2 -1626.593} C_VEL
LIN {X 0,Y 587.244,Z 638.33,A -85,B 0,C 180,E1 -1627.738,E2 -1627.738} C_VEL
LIN {X 0,Y 587.312,Z 629.899,A -85,B 0,C 180,E1 -1628.95,E2 -1628.95} C_VEL
LIN {X 0,Y 587.344,Z 621.14,A -85,B 0,C 180,E1 -1629.992,E2 -1629.992} C_VEL
LIN {X 0,Y 587.466,Z 610.496,A -85,B 0,C 180,E1 -1631.035,E2 -1631.035} C_VEL
LIN {X 0,Y 587.551,Z 599.748,A -85,B 0,C 180,E1 -1631.908,E2 -1631.908} C_VEL
LIN {X 0,Y 587.654,Z 588.006,A -85,B 0,C 180,E1 -1632.695,E2 -1632.695} C_VEL
LIN {X 0,Y 587.763,Z 575.037,A -85,B 0,C 180,E1 -1633.396,E2 -1633.396} C_VEL
LIN {X 0,Y 587.859,Z 563.544,A -85,B 0,C 180,E1 -1633.885,E2 -1633.885} C_VEL
LIN {X 0,Y 587.36,Z 558.077,A -85,B 0,C 180,E1 -1634.099,E2 -1634.099} C_VEL
LIN {X 0,Y 584.579,Z 549.214,A -85,B 0,C 180,E1 -1634.446,E2 -1634.446} C_VEL
LIN {X 0,Y 581.74,Z 540.171,A -85,B 0,C 180,E1 -1634.732,E2 -1634.732} C_VEL
LIN {X 0,Y 581.14,Z 534.428,A -85,B 0,C 180,E1 -1634.848,E2 -1634.848} C_VEL
LIN {X 0,Y 581.268,Z 401.194,A -85,B 0,C 180,E1 -1636.535,E2 -1636.535} C_VEL
LIN {X 0,Y 580.657,Z 397.547,A -85,B 0,C 180,E1 -1636.615,E2 -1636.615} C_VEL
LIN {X 0,Y 580.802,Z 376.006,A -85,B 0,C 180,E1 -1639.293,E2 -1639.293} C_VEL
LIN {X 0,Y 581.035,Z 354.59,A -85,B 0,C 180,E1 -1642.022,E2 -1642.022} C_VEL
LIN {X 0,Y 581.205,Z 338.654,A -85,B 0,C 180,E1 -1644.086,E2 -1644.086} C_VEL
LIN {X 0,Y 580.459,Z 333.789,A -85,B 0,C 180,E1 -1644.759,E2 -1644.759} C_VEL
LIN {X 0,Y 580.278,Z 332.904,A -85,B 0,C 180,E1 -1644.973,E2 -1644.973} C_VEL
LIN {X 0,Y 580.232,Z 332.837,A -85,B 0,C 180,E1 -1647.846,E2 -1647.846} C_VEL
LIN {X 0,Y 580.251,Z 332.828,A -85,B 0,C 180,E1 -1650.689,E2 -1650.689} C_VEL
LIN {X 0,Y 580.266,Z 332.825,A -85,B 0,C 180,E1 -1653.31,E2 -1653.31} C_VEL
LIN {X 0,Y 580.215,Z 332.836,A -85,B 0,C 180,E1 -1655.752,E2 -1655.752} C_VEL
LIN {X 0,Y 580.265,Z 332.833,A -85,B 0,C 180,E1 -1658.148,E2 -1658.148} C_VEL
LIN {X 0,Y 580.234,Z 332.828,A -85,B 0,C 180,E1 -1660.849,E2 -1660.849} C_VEL
LIN {X 0,Y 580.225,Z 332.831,A -85,B 0,C 180,E1 -1663.663,E2 -1663.663} C_VEL
LIN {X 0,Y 580.22,Z 332.83,A -85,B 0,C 180,E1 -1666.615,E2 -1666.615} C_VEL
LIN {X 0,Y 580.234,Z 332.828,A -85,B 0,C 180,E1 -1669.151,E2 -1669.151} C_VEL
LIN {X 0,Y 580.267,Z 332.832,A -85,B 0,C 180,E1 -1671.93,E2 -1671.93} C_VEL
LIN {X 0,Y 580.214,Z 332.835,A -85,B 0,C 180,E1 -1674.45,E2 -1674.45} C_VEL
LIN {X 0,Y 580.238,Z 332.828,A -85,B 0,C 180,E1 -1676.972,E2 -1676.972} C_VEL
LIN {X 0,Y 580.27,Z 332.826,A -85,B 0,C 180,E1 -1679.423,E2 -1679.423} C_VEL
LIN {X 0,Y 580.231,Z 332.839,A -85,B 0,C 180,E1 -1682.154,E2 -1682.154} C_VEL
LIN {X 0,Y 580.281,Z 333.005,A -85,B 0,C 180,E1 -1683.037,E2 -1683.037} C_VEL
LIN {X 0,Y 581.65,Z 339.317,A -85,B 0,C 180,E1 -1683.872,E2 -1683.872} C_VEL
LIN {X 0,Y 581.334,Z 361.792,A -85,B 0,C 180,E1 -1686.487,E2 -1686.487} C_VEL
LIN {X 0,Y 581.033,Z 387.879,A -85,B 0,C 180,E1 -1689.465,E2 -1689.465} C_VEL
LIN {X 0,Y 580.972,Z 398.632,A -85,B 0,C 180,E1 -1690.659,E2 -1690.659} C_VEL
LIN {X 0,Y 581.899,Z 404.262,A -85,B 0,C 180,E1 -1690.781,E2 -1690.781} C_VEL
LIN {X 0,Y 581.495,Z 563.797,A -85,B 0,C 180,E1 -1692.817,E2 -1692.817} C_VEL
LIN {X 0,Y 581.453,Z 578.212,A -85,B 0,C 180,E1 -1693.119,E2 -1693.119} C_VEL
LIN {X 0,Y 581.246,Z 593.558,A -85,B 0,C 180,E1 -1693.582,E2 -1693.582} C_VEL
LIN {X 0,Y 581.151,Z 606.805,A -85,B 0,C 180,E1 -1694.121,E2 -1694.121} C_VEL
LIN {X 0,Y 580.981,Z 619.263,A -85,B 0,C 180,E1 -1694.745,E2 -1694.745} C_VEL
LIN {X 0,Y 580.841,Z 631.108,A -85,B 0,C 180,E1 -1695.461,E2 -1695.461} C_VEL
LIN {X 0,Y 580.68,Z 643.417,A -85,B 0,C 180,E1 -1696.349,E2 -1696.349} C_VEL
LIN {X 0,Y 580.535,Z 655.706,A -85,B 0,C 180,E1 -1697.414,E2 -1697.414} C_VEL
LIN {X 0,Y 580.391,Z 665.955,A -85,B 0,C 180,E1 -1698.475,E2 -1698.475} C_VEL
LIN {X 0,Y 580.33,Z 674.651,A -85,B 0,C 180,E1 -1699.534,E2 -1699.534} C_VEL
LIN {X 0,Y 580.213,Z 683.253,A -85,B 0,C 180,E1 -1700.764,E2 -1700.764} C_VEL
LIN {X 0,Y 580.178,Z 690.392,A -85,B 0,C 180,E1 -1701.992,E2 -1701.992} C_VEL
LIN {X 0,Y 580.125,Z 697.085,A -85,B 0,C 180,E1 -1703.414,E2 -1703.414} C_VEL
LIN {X 0,Y 580.074,Z 702.169,A -85,B 0,C 180,E1 -1704.786,E2 -1704.786} C_VEL
LIN {X 0,Y 580.088,Z 705.165,A -85,B 0,C 180,E1 -1705.831,E2 -1705.831} C_VEL
LIN {X 0,Y 580.038,Z 708.118,A -85,B 0,C 180,E1 -1707.222,E2 -1707.222} C_VEL
LIN {X 0,Y 580.043,Z 709.887,A -85,B 0,C 180,E1 -1708.611,E2 -1708.611} C_VEL
LIN {X 0,Y 580.035,Z 710.496,A -85,B 0,C 180,E1 -1710,E2 -1710} C_VEL
LIN {X 0,Y 580.044,Z 709.955,A -85,B 0,C 180,E1 -1711.388,E2 -1711.388} C_VEL
LIN {X 0,Y 580.04,Z 708.261,A -85,B 0,C 180,E1 -1712.778,E2 -1712.778} C_VEL
LIN {X 0,Y 580.088,Z 705.395,A -85,B 0,C 180,E1 -1714.169,E2 -1714.169} C_VEL
LIN {X 0,Y 580.127,Z 701.331,A -85,B 0,C 180,E1 -1715.562,E2 -1715.562} C_VEL
LIN {X 0,Y 580.139,Z 695.918,A -85,B 0,C 180,E1 -1716.958,E2 -1716.958} C_VEL
LIN {X 0,Y 580.173,Z 688.985,A -85,B 0,C 180,E1 -1718.358,E2 -1718.358} C_VEL
LIN {X 0,Y 580.23,Z 681.558,A -85,B 0,C 180,E1 -1719.587,E2 -1719.587} C_VEL
LIN {X 0,Y 580.329,Z 672.82,A -85,B 0,C 180,E1 -1720.794,E2 -1720.794} C_VEL
LIN {X 0,Y 580.428,Z 661.937,A -85,B 0,C 180,E1 -1722.056,E2 -1722.056} C_VEL
LIN {X 0,Y 580.594,Z 650.856,A -85,B 0,C 180,E1 -1723.118,E2 -1723.118} C_VEL
LIN {X 0,Y 580.72,Z 639.928,A -85,B 0,C 180,E1 -1724.007,E2 -1724.007} C_VEL
LIN {X 0,Y 580.904,Z 628.338,A -85,B 0,C 180,E1 -1724.808,E2 -1724.808} C_VEL
LIN {X 0,Y 581.069,Z 614.278,A -85,B 0,C 180,E1 -1725.611,E2 -1725.611} C_VEL
LIN {X 0,Y 581.191,Z 599.415,A -85,B 0,C 180,E1 -1726.284,E2 -1726.284} C_VEL
LIN {X 0,Y 581.384,Z 584.533,A -85,B 0,C 180,E1 -1726.797,E2 -1726.797} C_VEL
LIN {X 0,Y 581.492,Z 568.537,A -85,B 0,C 180,E1 -1727.19,E2 -1727.19} C_VEL
LIN {X 0,Y 581.575,Z 546.9,A -85,B 0,C 180,E1 -1727.503,E2 -1727.503} C_VEL
LIN {X 0,Y 581.844,Z 403.242,A -85,B 0,C 180,E1 -1729.324,E2 -1729.324} C_VEL
LIN {X 0,Y 580.978,Z 398.631,A -85,B 0,C 180,E1 -1729.431,E2 -1729.431} C_VEL
LIN {X 0,Y 581.195,Z 373.991,A -85,B 0,C 180,E1 -1732.203,E2 -1732.203} C_VEL
LIN {X 0,Y 581.522,Z 349.519,A -85,B 0,C 180,E1 -1735.024,E2 -1735.024} C_VEL
LIN {X 0,Y 581.532,Z 338.226,A -85,B 0,C 180,E1 -1736.353,E2 -1736.353} C_VEL
LIN {X 0,Y 580.265,Z 332.977,A -85,B 0,C 180,E1 -1737.061,E2 -1737.061} C_VEL
LIN {X 0,Y 580.254,Z 332.832,A -85,B 0,C 180,E1 -1739.775,E2 -1739.775} C_VEL
LIN {X 0,Y 580.268,Z 332.831,A -85,B 0,C 180,E1 -1742.202,E2 -1742.202} C_VEL
LIN {X 0,Y 580.263,Z 332.826,A -85,B 0,C 180,E1 -1744.698,E2 -1744.698} C_VEL
LIN {X 0,Y 580.256,Z 332.827,A -85,B 0,C 180,E1 -1747.272,E2 -1747.272} C_VEL
LIN {X 0,Y 580.248,Z 332.831,A -85,B 0,C 180,E1 -1750.265,E2 -1750.265} C_VEL
LIN {X 0,Y 580.243,Z 332.827,A -85,B 0,C 180,E1 -1752.709,E2 -1752.709} C_VEL
LIN {X 0,Y 580.25,Z 332.832,A -85,B 0,C 180,E1 -1755.611,E2 -1755.611} C_VEL
LIN {X 0,Y 580.24,Z 332.831,A -85,B 0,C 180,E1 -1758.228,E2 -1758.228} C_VEL
LIN {X 0,Y 580.26,Z 332.824,A -85,B 0,C 180,E1 -1760.963,E2 -1760.963} C_VEL
LIN {X 0,Y 580.238,Z 332.835,A -85,B 0,C 180,E1 -1763.594,E2 -1763.594} C_VEL
LIN {X 0,Y 580.285,Z 332.825,A -85,B 0,C 180,E1 -1766.143,E2 -1766.143} C_VEL
LIN {X 0,Y 580.267,Z 332.823,A -85,B 0,C 180,E1 -1768.614,E2 -1768.614} C_VEL
LIN {X 0,Y 580.285,Z 332.823,A -85,B 0,C 180,E1 -1771.023,E2 -1771.023} C_VEL
LIN {X 0,Y 580.249,Z 332.829,A -85,B 0,C 180,E1 -1774.149,E2 -1774.149} C_VEL
LIN {X 0,Y 580.269,Z 332.823,A -85,B 0,C 180,E1 -1776.442,E2 -1776.442} C_VEL
LIN {X 0,Y 580.269,Z 332.829,A -85,B 0,C 180,E1 -1779.437,E2 -1779.437} C_VEL
LIN {X 0,Y 580.254,Z 332.834,A -85,B 0,C 180,E1 -1781.645,E2 -1781.645} C_VEL
LIN {X 0,Y 580.261,Z 332.83,A -85,B 0,C 180,E1 -1783.825,E2 -1783.825} C_VEL
LIN {X 0,Y 580.322,Z 332.82,A -85,B 0,C 180,E1 -1785.983,E2 -1785.983} C_VEL
LIN {X 0,Y 580.307,Z 332.818,A -85,B 0,C 180,E1 -1788.827,E2 -1788.827} C_VEL
LIN {X 0,Y 580.325,Z 332.824,A -85,B 0,C 180,E1 -1791.644,E2 -1791.644} C_VEL
LIN {X 0,Y 580.282,Z 332.826,A -85,B 0,C 180,E1 -1793.742,E2 -1793.742} C_VEL
LIN {X 0,Y 580.271,Z 332.826,A -85,B 0,C 180,E1 -1795.833,E2 -1795.833} C_VEL
LIN {X 0,Y 580.344,Z 332.817,A -85,B 0,C 180,E1 -1797.918,E2 -1797.918} C_VEL
LIN {X 0,Y 580.347,Z 332.813,A -85,B 0,C 180,E1 -1800.694,E2 -1800.694} C_VEL
LIN {X 0,Y 580.282,Z 332.831,A -85,B 0,C 180,E1 -1803.472,E2 -1803.472} C_VEL
LIN {X 0,Y 580.329,Z 332.822,A -85,B 0,C 180,E1 -1805.56,E2 -1805.56} C_VEL
LIN {X 0,Y 580.311,Z 332.816,A -85,B 0,C 180,E1 -1808.356,E2 -1808.356} C_VEL
LIN {X 0,Y 580.302,Z 332.827,A -85,B 0,C 180,E1 -1811.191,E2 -1811.191} C_VEL
LIN {X 0,Y 580.318,Z 332.816,A -85,B 0,C 180,E1 -1814.017,E2 -1814.017} C_VEL
LIN {X 0,Y 580.314,Z 332.822,A -85,B 0,C 180,E1 -1816.914,E2 -1816.914} C_VEL
LIN {X 0,Y 580.287,Z 332.821,A -85,B 0,C 180,E1 -1819.823,E2 -1819.823} C_VEL
LIN {X 0,Y 580.271,Z 332.823,A -85,B 0,C 180,E1 -1822.053,E2 -1822.053} C_VEL
LIN {X 0,Y 580.306,Z 332.827,A -85,B 0,C 180,E1 -1825.08,E2 -1825.08} C_VEL
LIN {X 0,Y 580.297,Z 332.82,A -85,B 0,C 180,E1 -1828.186,E2 -1828.186} C_VEL
LIN {X 0,Y 580.288,Z 332.823,A -85,B 0,C 180,E1 -1830.695,E2 -1830.695} C_VEL
LIN {X 0,Y 580.303,Z 332.825,A -85,B 0,C 180,E1 -1833.316,E2 -1833.316} C_VEL
LIN {X 0,Y 580.246,Z 332.827,A -85,B 0,C 180,E1 -1835.756,E2 -1835.756} C_VEL
LIN {X 0,Y 580.29,Z 332.82,A -85,B 0,C 180,E1 -1838.146,E2 -1838.146} C_VEL
LIN {X 0,Y 580.3,Z 332.822,A -85,B 0,C 180,E1 -1840.843,E2 -1840.843} C_VEL
LIN {X 0,Y 580.279,Z 332.824,A -85,B 0,C 180,E1 -1843.658,E2 -1843.658} C_VEL
LIN {X 0,Y 580.277,Z 332.824,A -85,B 0,C 180,E1 -1846.609,E2 -1846.609} C_VEL
LIN {X 0,Y 580.3,Z 332.827,A -85,B 0,C 180,E1 -1849.157,E2 -1849.157} C_VEL
LIN {X 0,Y 580.291,Z 332.821,A -85,B 0,C 180,E1 -1851.927,E2 -1851.927} C_VEL
LIN {X 0,Y 580.252,Z 332.829,A -85,B 0,C 180,E1 -1854.453,E2 -1854.453} C_VEL
LIN {X 0,Y 580.29,Z 332.83,A -85,B 0,C 180,E1 -1856.975,E2 -1856.975} C_VEL
LIN {X 0,Y 580.302,Z 332.823,A -85,B 0,C 180,E1 -1859.426,E2 -1859.426} C_VEL
LIN {X 0,Y 580.297,Z 332.821,A -85,B 0,C 180,E1 -1862.142,E2 -1862.142} C_VEL
LIN {X 0,Y 580.354,Z 333.052,A -85,B 0,C 180,E1 -1863.797,E2 -1863.797} C_VEL
LIN {X 0,Y 581.601,Z 338.02,A -85,B 0,C 180,E1 -1864.406,E2 -1864.406} C_VEL
LIN {X 0,Y 581.453,Z 357.816,A -85,B 0,C 180,E1 -1866.493,E2 -1866.493} C_VEL
LIN {X 0,Y 581.14,Z 384.81,A -85,B 0,C 180,E1 -1869.284,E2 -1869.284} C_VEL
LIN {X 0,Y 581.045,Z 397.965,A -85,B 0,C 180,E1 -1870.609,E2 -1870.609} C_VEL
LIN {X 0,Y 581.931,Z 404.159,A -85,B 0,C 180,E1 -1870.735,E2 -1870.735} C_VEL
LIN {X 0,Y 581.526,Z 564.891,A -85,B 0,C 180,E1 -1872.787,E2 -1872.787} C_VEL
LIN {X 0,Y 581.411,Z 580.709,A -85,B 0,C 180,E1 -1873.136,E2 -1873.136} C_VEL
LIN {X 0,Y 581.238,Z 596.044,A -85,B 0,C 180,E1 -1873.628,E2 -1873.628} C_VEL
LIN {X 0,Y 581.123,Z 609.769,A -85,B 0,C 180,E1 -1874.21,E2 -1874.21} C_VEL
LIN {X 0,Y 580.942,Z 623.242,A -85,B 0,C 180,E1 -1874.924,E2 -1874.924} C_VEL
LIN {X 0,Y 580.804,Z 636.48,A -85,B 0,C 180,E1 -1875.783,E2 -1875.783} C_VEL
LIN {X 0,Y 580.608,Z 648.289,A -85,B 0,C 180,E1 -1876.704,E2 -1876.704} C_VEL
LIN {X 0,Y 580.479,Z 659.749,A -85,B 0,C 180,E1 -1877.768,E2 -1877.768} C_VEL
LIN {X 0,Y 580.307,Z 670.455,A -85,B 0,C 180,E1 -1878.954,E2 -1878.954} C_VEL
LIN {X 0,Y 580.269,Z 678.857,A -85,B 0,C 180,E1 -1880.062,E2 -1880.062} C_VEL
LIN {X 0,Y 580.213,Z 686.733,A -85,B 0,C 180,E1 -1881.291,E2 -1881.291} C_VEL
LIN {X 0,Y 580.13,Z 694.089,A -85,B 0,C 180,E1 -1882.692,E2 -1882.692} C_VEL
LIN {X 0,Y 580.131,Z 699.924,A -85,B 0,C 180,E1 -1884.09,E2 -1884.09} C_VEL
LIN {X 0,Y 580.041,Z 703.385,A -85,B 0,C 180,E1 -1885.135,E2 -1885.135} C_VEL
LIN {X 0,Y 580.105,Z 706.888,A -85,B 0,C 180,E1 -1886.527,E2 -1886.527} C_VEL
LIN {X 0,Y 580.038,Z 709.193,A -85,B 0,C 180,E1 -1887.917,E2 -1887.917} C_VEL
LIN {X 0,Y 580.036,Z 710.349,A -85,B 0,C 180,E1 -1889.306,E2 -1889.306} C_VEL
LIN {X 0,Y 580.036,Z 710.349,A -85,B 0,C 180,E1 -1890.694,E2 -1890.694} C_VEL
LIN {X 0,Y 580.038,Z 709.192,A -85,B 0,C 180,E1 -1892.083,E2 -1892.083} C_VEL
LIN {X 0,Y 580.105,Z 706.886,A -85,B 0,C 180,E1 -1893.473,E2 -1893.473} C_VEL
LIN {X 0,Y 580.041,Z 703.384,A -85,B 0,C 180,E1 -1894.865,E2 -1894.865} C_VEL
LIN {X 0,Y 580.092,Z 698.608,A -85,B 0,C 180,E1 -1896.26,E2 -1896.26} C_VEL
LIN {X 0,Y 580.165,Z 692.423,A -85,B 0,C 180,E1 -1897.658,E2 -1897.658} C_VEL
LIN {X 0,Y 580.207,Z 684.649,A -85,B 0,C 180,E1 -1899.06,E2 -1899.06} C_VEL
LIN {X 0,Y 580.309,Z 676.368,A -85,B 0,C 180,E1 -1900.29,E2 -1900.29} C_VEL
LIN {X 0,Y 580.383,Z 666.394,A -85,B 0,C 180,E1 -1901.525,E2 -1901.525} C_VEL
LIN {X 0,Y 580.541,Z 656.188,A -85,B 0,C 180,E1 -1902.586,E2 -1902.586} C_VEL
LIN {X 0,Y 580.678,Z 644.017,A -85,B 0,C 180,E1 -1903.651,E2 -1903.651} C_VEL
LIN {X 0,Y 580.846,Z 631.803,A -85,B 0,C 180,E1 -1904.542,E2 -1904.542} C_VEL
LIN {X 0,Y 580.971,Z 618.516,A -85,B 0,C 180,E1 -1905.345,E2 -1905.345} C_VEL
LIN {X 0,Y 581.192,Z 603.832,A -85,B 0,C 180,E1 -1906.058,E2 -1906.058} C_VEL
LIN {X 0,Y 581.337,Z 589.612,A -85,B 0,C 180,E1 -1906.596,E2 -1906.596} C_VEL
LIN {X 0,Y 581.448,Z 574.401,A -85,B 0,C 180,E1 -1907.021,E2 -1907.021} C_VEL
LIN {X 0,Y 581.541,Z 559.134,A -85,B 0,C 180,E1 -1907.3,E2 -1907.3} C_VEL
LIN {X 0,Y 581.862,Z 402.559,A -85,B 0,C 180,E1 -1909.288,E2 -1909.288} C_VEL
LIN {X 0,Y 581.046,Z 397.961,A -85,B 0,C 180,E1 -1909.392,E2 -1909.392} C_VEL
LIN {X 0,Y 581.32,Z 370.411,A -85,B 0,C 180,E1 -1912.198,E2 -1912.198} C_VEL
LIN {X 0,Y 581.698,Z 341.617,A -85,B 0,C 180,E1 -1915.207,E2 -1915.207} C_VEL
LIN {X 0,Y 581.6,Z 338.018,A -85,B 0,C 180,E1 -1915.595,E2 -1915.595} C_VEL
LIN {X 0,Y 580.33,Z 332.941,A -85,B 0,C 180,E1 -1916.234,E2 -1916.234} C_VEL
LIN {X 0,Y 580.302,Z 332.828,A -85,B 0,C 180,E1 -1919.31,E2 -1919.31} C_VEL
LIN {X 0,Y 580.298,Z 332.822,A -85,B 0,C 180,E1 -1922.201,E2 -1922.201} C_VEL
LIN {X 0,Y 580.292,Z 332.828,A -85,B 0,C 180,E1 -1924.696,E2 -1924.696} C_VEL
LIN {X 0,Y 580.3,Z 332.825,A -85,B 0,C 180,E1 -1927.269,E2 -1927.269} C_VEL
LIN {X 0,Y 580.292,Z 332.824,A -85,B 0,C 180,E1 -1930.271,E2 -1930.271} C_VEL
LIN {X 0,Y 580.273,Z 332.833,A -85,B 0,C 180,E1 -1932.707,E2 -1932.707} C_VEL
LIN {X 0,Y 580.259,Z 332.826,A -85,B 0,C 180,E1 -1935.61,E2 -1935.61} C_VEL
LIN {X 0,Y 580.275,Z 332.829,A -85,B 0,C 180,E1 -1938.231,E2 -1938.231} C_VEL
LIN {X 0,Y 580.268,Z 332.827,A -85,B 0,C 180,E1 -1940.964,E2 -1940.964} C_VEL
LIN {X 0,Y 580.244,Z 332.828,A -85,B 0,C 180,E1 -1943.595,E2 -1943.595} C_VEL
LIN {X 0,Y 580.308,Z 332.827,A -85,B 0,C 180,E1 -1946.145,E2 -1946.145} C_VEL
LIN {X 0,Y 580.266,Z 332.83,A -85,B 0,C 180,E1 -1948.614,E2 -1948.614} C_VEL
LIN {X 0,Y 580.244,Z 332.829,A -85,B 0,C 180,E1 -1951.021,E2 -1951.021} C_VEL
LIN {X 0,Y 580.253,Z 332.833,A -85,B 0,C 180,E1 -1953.674,E2 -1953.674} C_VEL
LIN {X 0,Y 580.29,Z 333.027,A -85,B 0,C 180,E1 -1955.193,E2 -1955.193} C_VEL
LIN {X 0,Y 581.222,Z 337.968,A -85,B 0,C 180,E1 -1955.915,E2 -1955.915} C_VEL
LIN {X 0,Y 580.994,Z 356.792,A -85,B 0,C 180,E1 -1958.35,E2 -1958.35} C_VEL
LIN {X 0,Y 580.795,Z 378.506,A -85,B 0,C 180,E1 -1961.114,E2 -1961.114} C_VEL
LIN {X 0,Y 580.669,Z 397.591,A -85,B 0,C 180,E1 -1963.475,E2 -1963.475} C_VEL
LIN {X 0,Y 581.414,Z 403.419,A -85,B 0,C 180,E1 -1963.588,E2 -1963.588} C_VEL
LIN {X 0,Y 581.142,Z 535.923,A -85,B 0,C 180,E1 -1965.266,E2 -1965.266} C_VEL
LIN {X 0,Y 581.052,Z 550.171,A -85,B 0,C 180,E1 -1965.591,E2 -1965.591} C_VEL
LIN {X 0,Y 580.944,Z 563.704,A -85,B 0,C 180,E1 -1966.043,E2 -1966.043} C_VEL
LIN {X 0,Y 580.803,Z 576.746,A -85,B 0,C 180,E1 -1966.619,E2 -1966.619} C_VEL
LIN {X 0,Y 580.679,Z 589.403,A -85,B 0,C 180,E1 -1967.328,E2 -1967.328} C_VEL
LIN {X 0,Y 580.545,Z 600.864,A -85,B 0,C 180,E1 -1968.124,E2 -1968.124} C_VEL
LIN {X 0,Y 580.463,Z 611.468,A -85,B 0,C 180,E1 -1969.008,E2 -1969.008} C_VEL
LIN {X 0,Y 580.313,Z 621.899,A -85,B 0,C 180,E1 -1970.062,E2 -1970.062} C_VEL
LIN {X 0,Y 580.254,Z 630.572,A -85,B 0,C 180,E1 -1971.116,E2 -1971.116} C_VEL
LIN {X 0,Y 580.177,Z 638.825,A -85,B 0,C 180,E1 -1972.343,E2 -1972.343} C_VEL
LIN {X 0,Y 580.124,Z 644.749,A -85,B 0,C 180,E1 -1973.416,E2 -1973.416} C_VEL
LIN {X 0,Y 580.077,Z 650.775,A -85,B 0,C 180,E1 -1974.787,E2 -1974.787} C_VEL
LIN {X 0,Y 580.103,Z 654.299,A -85,B 0,C 180,E1 -1975.832,E2 -1975.832} C_VEL
LIN {X 0,Y 580.041,Z 657.748,A -85,B 0,C 180,E1 -1977.222,E2 -1977.222} C_VEL
LIN {X 0,Y 580.045,Z 659.772,A -85,B 0,C 180,E1 -1978.612,E2 -1978.612} C_VEL
LIN {X 0,Y 580.037,Z 660.496,A -85,B 0,C 180,E1 -1980,E2 -1980} C_VEL
LIN {X 0,Y 580.042,Z 659.858,A -85,B 0,C 180,E1 -1981.389,E2 -1981.389} C_VEL
LIN {X 0,Y 580.039,Z 657.93,A -85,B 0,C 180,E1 -1982.778,E2 -1982.778} C_VEL
LIN {X 0,Y 580.104,Z 654.571,A -85,B 0,C 180,E1 -1984.169,E2 -1984.169} C_VEL
LIN {X 0,Y 580.128,Z 649.763,A -85,B 0,C 180,E1 -1985.562,E2 -1985.562} C_VEL
LIN {X 0,Y 580.137,Z 645.148,A -85,B 0,C 180,E1 -1986.596,E2 -1986.596} C_VEL
LIN {X 0,Y 580.173,Z 638.322,A -85,B 0,C 180,E1 -1987.833,E2 -1987.833} C_VEL
LIN {X 0,Y 580.261,Z 629.892,A -85,B 0,C 180,E1 -1989.059,E2 -1989.059} C_VEL
LIN {X 0,Y 580.324,Z 621.138,A -85,B 0,C 180,E1 -1990.114,E2 -1990.114} C_VEL
LIN {X 0,Y 580.453,Z 610.491,A -85,B 0,C 180,E1 -1991.17,E2 -1991.17} C_VEL
LIN {X 0,Y 580.58,Z 599.742,A -85,B 0,C 180,E1 -1992.053,E2 -1992.053} C_VEL
LIN {X 0,Y 580.696,Z 587.99,A -85,B 0,C 180,E1 -1992.849,E2 -1992.849} C_VEL
LIN {X 0,Y 580.853,Z 575.024,A -85,B 0,C 180,E1 -1993.558,E2 -1993.558} C_VEL
LIN {X 0,Y 580.99,Z 561.802,A -85,B 0,C 180,E1 -1994.12,E2 -1994.12} C_VEL
LIN {X 0,Y 581.066,Z 547.799,A -85,B 0,C 180,E1 -1994.562,E2 -1994.562} C_VEL
